(* CoDeSys 2.3.9.41 project: plc_12.pro *)
(* Libraries: STANDARD.LIB 4.10.05 13:14:46, IECSFC.LIB 13.4.06 17:51:28, SYSLIBTIME.LIB 20.2.06 15:31:16, SYSTASKINFO.LIB 20.2.06 15:31:38, ANALYZATION.LIB 5.10.99 11:05:06, SYSLIBCALLBACK.LIB 20.2.06 15:31:08, Util.lib 18.5.10 17:14:28 *)

(* PLC configuration (modules and I/O channels)
Fast discrete inputs [I_SIMPLE_INPUT] node 0, in %IB0 out %QB0 {ChannellName = Fast discrete inputs; Filtrationtime = 1}
  AT %IX0.0 [BitInput] Discrete input 1 {ChannellName = Enter name}
  AT %IX0.1 [BitInput] Discrete input 2 {ChannellName = Enter name}
  AT %IX0.2 [BitInput] Discrete input 3 {ChannellName = Enter name}
  CONTR_PHASE AT %IX0.3 [BitInput] Discrete input 4 {ChannellName = Enter name}
Discrete inputs [ID130] node 1, in %IB1 out %QB1 {ChannellName = Discrete inputs; Filtrationtime_GeneralINP = 0; PinCount = 32}
  AT %IB1.0 [ByteInput] 8 discrete inputs {ChannellName = Enter name}
  AT %IB1.1 [ByteInput] 8 discrete inputs {ChannellName = Enter name}
  AT %IB1.2 [ByteInput] 8 discrete inputs {ChannellName = Enter name}
  AT %IB1.3 [ByteInput] 8 discrete inputs {ChannellName = Enter name}
Fast discrete outputs [OWEN_ID570] node 2, in %IB2 out %QB2 {ChannellName = Fast discrete outputs; SafeValueBool = FALSE; SafeValueBool = FALSE; SafeValueBool = FALSE; SafeValueBool = FALSE; Visibility = No}
  ELV_DROB_RUN AT %QX2.0 [BitOutput] Fast discrete output 1 {ChannellName = Enter name}
  DROB_SHOK_1 AT %QX2.1 [BitOutput] Fast discrete output 2 {ChannellName = Enter name}
  DROB_SHOK_2 AT %QX2.2 [BitOutput] Fast discrete output 3 {ChannellName = Enter name}
  CONV_DROB AT %QX2.3 [BitOutput] Fast discrete output 4 {ChannellName = Enter name}
Discrete outputs [ID131] node 3, in %IB3 out %QB3 {ChannellName = Discrete outputs; SafeValueByte = 0; SafeValueByte = 0; SafeValueByteM = 0; PinCount = 24}
  AT %QB3.0 [ByteOutput] 8 discrete outputs {ChannellName = Enter name}
  AT %QB3.1 [ByteOutput] 8 discrete outputs {ChannellName = Enter name}
  AT %QB3.2 [ByteOutput] 4 discrete outputs {ChannellName = Enter name}
Special input [ID103] node 4, in %IB4 out %QB4 {ChannellName = Special input}
  AT %IX4.0 [BitInput] Special input {ChannellName = Enter name}
Special output [ID104] node 5, in %IB5 out %QB5 {ChannellName = Special output}
  AT %QX5.0 [BitOutput] Special output {ChannellName = Enter name}
AT %QD6.0 [DWordOutput] Last address {ChannellName = Enter name}
AT %QW6.1 [WordOutput] Last error {ChannellName = Enter name}
RS-485-1 [COM1_USART] node 0, in %IB6.0 out %QB6.0 {ChannellName = RS-485-1; CommunicationSpeed = 115200; Parity = NO PARITY CHECK; BitLength = 8 bits; StopLength = One stop bit; InterfaceType = RS485; FrameOriented = RTU; Timeout = 0; Visibility = No}
Universal Modbus device [ID2000] node 1, in %IB6.1 out %QB6.1 {ChannellName = Universal Modbus device; ModuleIP = 10:0:0:223; ServiceTimeout = 150; TCPport = 502; NetMode = Serial; ModuleSlaveAddress = 8; RequestType = By poll time; PeriodOfService = 10; Visibility = No; RepeatCounter = 0; ByteSequence = Trace_mode}
  AT %QB6.1.0 [ComChannel] Command (0xff - Start) {ChannellName = Enter name}
MV8_0 AT %QW6.1.0.0 [WordOutput] {ChannellName = Enter name}
MV8_1 AT %QW6.1.1.0 [WordOutput] {ChannellName = Enter name}
Universal Modbus device [ID2000] node 2, in %IB6.2 out %QB6.2 {ChannellName = Universal Modbus device; ModuleIP = 10:0:0:223; ServiceTimeout = 150; TCPport = 502; NetMode = Serial; ModuleSlaveAddress = 16; RequestType = By poll time; PeriodOfService = 10; Visibility = No; RepeatCounter = 0; ByteSequence = Trace_mode}
  AT %QB6.2.0 [ComChannel] Command (0xff - Start) {ChannellName = Enter name}
MV16_0 AT %QW6.2.0.0 [WordOutput] {ChannellName = Enter name}
MV16_1 AT %QW6.2.1.0 [WordOutput] {ChannellName = Enter name}
Universal Modbus device [ID2000] node 3, in %IB6.3 out %QB6.3 {ChannellName = Universal Modbus device; ModuleIP = 10:0:0:223; ServiceTimeout = 150; TCPport = 502; NetMode = Serial; ModuleSlaveAddress = 24; RequestType = By poll time; PeriodOfService = 10; Visibility = No; RepeatCounter = 0; ByteSequence = Trace_mode}
  AT %QB6.3.0 [ComChannel] Command (0xff - Start) {ChannellName = Enter name}
MV24_0 AT %QW6.3.0.0 [WordOutput] {ChannellName = Enter name}
MV24_1 AT %QW6.3.1.0 [WordOutput] {ChannellName = Enter name}
Universal Modbus device [ID2000] node 4, in %IB6.4 out %QB6.4 {ChannellName = Universal Modbus device; ModuleIP = 10:0:0:223; ServiceTimeout = 150; TCPport = 502; NetMode = Serial; ModuleSlaveAddress = 32; RequestType = By poll time; PeriodOfService = 10; Visibility = No; RepeatCounter = 0; ByteSequence = Trace_mode}
  AT %QB6.4.0 [ComChannel] Command (0xff - Start) {ChannellName = Enter name}
MU01 AT %QW6.4.0.0 [WordOutput] {ChannellName = Enter name}
MU02 AT %QW6.4.1.0 [WordOutput] {ChannellName = Enter name}
MU03 AT %QW6.4.2.0 [WordOutput] {ChannellName = Enter name}
MU04 AT %QW6.4.3.0 [WordOutput] {ChannellName = Enter name}
MU05 AT %QW6.4.4.0 [WordOutput] {ChannellName = Enter name}
MU06 AT %QW6.4.5.0 [WordOutput] {ChannellName = Enter name}
MU07 AT %QW6.4.6.0 [WordOutput] {ChannellName = Enter name}
MU08 AT %QW6.4.7.0 [WordOutput] {ChannellName = Enter name}
MU09 AT %QW6.4.8.0 [WordOutput] {ChannellName = Enter name}
MU10 AT %QW6.4.9.0 [WordOutput] {ChannellName = Enter name}
MU11 AT %QW6.4.10.0 [WordOutput] {ChannellName = Enter name}
MU12 AT %QW6.4.11.0 [WordOutput] {ChannellName = Enter name}
MU13 AT %QW6.4.12.0 [WordOutput] {ChannellName = Enter name}
MU14 AT %QW6.4.13.0 [WordOutput] {ChannellName = Enter name}
MU15 AT %QW6.4.14.0 [WordOutput] {ChannellName = Enter name}
MU16 AT %QW6.4.15.0 [WordOutput] {ChannellName = Enter name}
MU17 AT %QW6.4.16.0 [WordOutput] {ChannellName = Enter name}
MU18 AT %QW6.4.17.0 [WordOutput] {ChannellName = Enter name}
MU19 AT %QW6.4.18.0 [WordOutput] {ChannellName = Enter name}
MU20 AT %QW6.4.19.0 [WordOutput] {ChannellName = Enter name}
MU21 AT %QW6.4.20.0 [WordOutput] {ChannellName = Enter name}
%MMU22 AT %QW6.4.21.0 [WordOutput] {ChannellName = Enter name}
MU23 AT %QW6.4.22.0 [WordOutput] {ChannellName = Enter name}
MU24 AT %QW6.4.23.0 [WordOutput] {ChannellName = Enter name}
MU25 AT %QW6.4.24.0 [WordOutput] {ChannellName = Enter name}
MU26 AT %QW6.4.25.0 [WordOutput] {ChannellName = Enter name}
MU27 AT %QW6.4.26.0 [WordOutput] {ChannellName = Enter name}
MU28 AT %QW6.4.27.0 [WordOutput] {ChannellName = Enter name}
MU29 AT %QW6.4.28.0 [WordOutput] {ChannellName = Enter name}
MU30 AT %QW6.4.29.0 [WordOutput] {ChannellName = Enter name}
MU31 AT %QW6.4.30.0 [WordOutput] {ChannellName = Enter name}
MU32 AT %QW6.4.31.0 [WordOutput] {ChannellName = Enter name}
AT %QB6.5.0 [ComChannel] Command (0xff - Start) {ChannellName = Enter name}
ELV_CURRENT_4 AT %QW6.5.0.0 [WordOutput] {ChannellName = Enter name}
SHNK_CURRENT_4 AT %QW6.5.1.0 [WordOutput] {ChannellName = Enter name}
MILL_SUCTION_4 AT %QW6.5.2.0 [WordOutput] {ChannellName = Enter name}
SHNK_CURRENT_3 AT %QW6.5.3.0 [WordOutput] {ChannellName = Enter name}
MILL_SUCTION_3 AT %QW6.5.4.0 [WordOutput] {ChannellName = Enter name}
TCP [TCP_ID221] node 0, in %IB7.0.0 out %QB7.0.0 {ChannellName = TCP; RemotePort = 502; Visibility = No}
TCP [TCP_ID221] node 1, in %IB7.0.1 out %QB7.0.1 {ChannellName = TCP; RemotePort = 503; Visibility = No}
CONV_1_DIO AT %QW7.1.0 [WordOutput] {ChannellName = Enter name}
CONV_1_CURRENT AT %QW7.2.0 [WordOutput] {ChannellName = Enter name}
CONV_1_FREQ AT %QW7.3.0 [WordOutput] {ChannellName = Enter name}
CONV_1_SETPOINT AT %QW7.4.0 [WordOutput] {ChannellName = Enter name}
CONV_1_wHOUR AT %QW7.5.0 [WordOutput] {ChannellName = Enter name}
CONV_1_stopTIME AT %QW7.6.0 [WordOutput] {ChannellName = Enter name}
CONV_1_startTIME AT %QW7.7.0 [WordOutput] {ChannellName = Enter name}
CONV_1_stopTIME_W AT %QW7.8.0 [WordOutput] {ChannellName = Enter name}
CONV_1_startTIME_W AT %QW7.9.0 [WordOutput] {ChannellName = Enter name}
FAN_1_DIO AT %QW7.10.0 [WordOutput] {ChannellName = Enter name}
FAN_1_CURRENT AT %QW7.11.0 [WordOutput] {ChannellName = Enter name}
FAN_1_FREQ AT %QW7.12.0 [WordOutput] {ChannellName = Enter name}
FAN_1_SETPOINT AT %QW7.13.0 [WordOutput] {ChannellName = Enter name}
FAN_1_SUCTION AT %QW7.14.0 [WordOutput] {ChannellName = Enter name}
FAN_1_wHOUR AT %QW7.15.0 [WordOutput] {ChannellName = Enter name}
FAN_1_stopTIME AT %QW7.16.0 [WordOutput] {ChannellName = Enter name}
FAN_1_startTIME AT %QW7.17.0 [WordOutput] {ChannellName = Enter name}
FAN_1_stopTIME_W AT %QW7.18.0 [WordOutput] {ChannellName = Enter name}
FAN_1_startTIME_W AT %QW7.19.0 [WordOutput] {ChannellName = Enter name}
MILL_1_DIO AT %QW7.20.0 [WordOutput] {ChannellName = Enter name}
MILL_1_CURRENT AT %QW7.21.0 [WordOutput] {ChannellName = Enter name}
MILL_1_FREQ AT %QW7.22.0 [WordOutput] {ChannellName = Enter name}
MILL_1_SETPOINT AT %QW7.23.0 [WordOutput] {ChannellName = Enter name}
MILL_1_wHOUR AT %QW7.24.0 [WordOutput] {ChannellName = Enter name}
MILL_1_stopTIME AT %QW7.25.0 [WordOutput] {ChannellName = Enter name}
MILL_1_startTIME AT %QW7.26.0 [WordOutput] {ChannellName = Enter name}
MILL_1_stopTIME_W AT %QW7.27.0 [WordOutput] {ChannellName = Enter name}
MILL_1_startTIME_W AT %QW7.28.0 [WordOutput] {ChannellName = Enter name}
SEP_1_DIO AT %QW7.29.0 [WordOutput] {ChannellName = Enter name}
SEP_1_CURRENT AT %QW7.30.0 [WordOutput] {ChannellName = Enter name}
SEP_1_FREQ AT %QW7.31.0 [WordOutput] {ChannellName = Enter name}
SEP_1_SETPOINT AT %QW7.32.0 [WordOutput] {ChannellName = Enter name}
SEP_1_wHOUR AT %QW7.33.0 [WordOutput] {ChannellName = Enter name}
SEP_1_stopTIME AT %QW7.34.0 [WordOutput] {ChannellName = Enter name}
SEP_1_startTIME AT %QW7.35.0 [WordOutput] {ChannellName = Enter name}
SEP_1_stopTIME_W AT %QW7.36.0 [WordOutput] {ChannellName = Enter name}
SEP_1_startTIME_W AT %QW7.37.0 [WordOutput] {ChannellName = Enter name}
2 byte [Register] node 38, in %IB7.38 out %QB7.38 {ChannellName = 2 byte}
  CONV_2_DIO AT %QW7.38.0 [WordOutput] {ChannellName = Enter name}
2 byte [Register] node 39, in %IB7.39 out %QB7.39 {ChannellName = 2 byte}
  CONV_2_CURRENT AT %QW7.39.0 [WordOutput] {ChannellName = Enter name}
2 byte [Register] node 40, in %IB7.40 out %QB7.40 {ChannellName = 2 byte}
  CONV_2_FREQ AT %QW7.40.0 [WordOutput] {ChannellName = Enter name}
2 byte [Register] node 41, in %IB7.41 out %QB7.41 {ChannellName = 2 byte}
  CONV_2_SETPOINT AT %QW7.41.0 [WordOutput] {ChannellName = Enter name}
  CONV_2_wHOUR AT %QW7.42.0 [WordOutput] {ChannellName = Enter name}
  CONV_2_stopTIME AT %QW7.43.0 [WordOutput] {ChannellName = Enter name}
  CONV_2_startTIME AT %QW7.44.0 [WordOutput] {ChannellName = Enter name}
  CONV_2_stopTIME_W AT %QW7.45.0 [WordOutput] {ChannellName = Enter name}
2 byte [Register] node 46, in %IB7.46 out %QB7.46 {ChannellName = 2 byte}
  CONV_2_startTIME_W AT %QW7.46.0 [WordOutput] {ChannellName = Enter name}
2 byte [Register] node 47, in %IB7.47 out %QB7.47 {ChannellName = 2 byte}
  FAN_2_DIO AT %QW7.47.0 [WordOutput] {ChannellName = Enter name}
2 byte [Register] node 48, in %IB7.48 out %QB7.48 {ChannellName = 2 byte}
  FAN_2_CURRENT AT %QW7.48.0 [WordOutput] {ChannellName = Enter name}
2 byte [Register] node 49, in %IB7.49 out %QB7.49 {ChannellName = 2 byte}
  FAN_2_FREQ AT %QW7.49.0 [WordOutput] {ChannellName = Enter name}
  FAN_2_SETPOINT AT %QW7.50.0 [WordOutput] {ChannellName = Enter name}
  FAN_2_SUCTION AT %QW7.51.0 [WordOutput] {ChannellName = Enter name}
  FAN_2_wHOUR AT %QW7.52.0 [WordOutput] {ChannellName = Enter name}
  FAN_2_stopTIME AT %QW7.53.0 [WordOutput] {ChannellName = Enter name}
  FAN_2_startTIME AT %QW7.54.0 [WordOutput] {ChannellName = Enter name}
2 byte [Register] node 55, in %IB7.55 out %QB7.55 {ChannellName = 2 byte}
  FAN_2_stopTIME_W AT %QW7.55.0 [WordOutput] {ChannellName = Enter name}
  FAN_2_startTIME_W AT %QW7.56.0 [WordOutput] {ChannellName = Enter name}
2 byte [Register] node 57, in %IB7.57 out %QB7.57 {ChannellName = 2 byte}
  MILL_2_DIO AT %QW7.57.0 [WordOutput] {ChannellName = Enter name}
  MILL_2_CURRENT AT %QW7.58.0 [WordOutput] {ChannellName = Enter name}
  MILL_2_FREQ AT %QW7.59.0 [WordOutput] {ChannellName = Enter name}
  MILL_2_SETPOINT AT %QW7.60.0 [WordOutput] {ChannellName = Enter name}
2 byte [Register] node 61, in %IB7.61 out %QB7.61 {ChannellName = 2 byte}
  MILL_2_wHOUR AT %QW7.61.0 [WordOutput] {ChannellName = Enter name}
  MILL_2_stopTIME AT %QW7.62.0 [WordOutput] {ChannellName = Enter name}
2 byte [Register] node 63, in %IB7.63 out %QB7.63 {ChannellName = 2 byte}
  MILL_2_startTIME AT %QW7.63.0 [WordOutput] {ChannellName = Enter name}
  MILL_2_stopTIME_W AT %QW7.64.0 [WordOutput] {ChannellName = Enter name}
2 byte [Register] node 65, in %IB7.65 out %QB7.65 {ChannellName = 2 byte}
  MILL_2_startTIME_W AT %QW7.65.0 [WordOutput] {ChannellName = Enter name}
2 byte [Register] node 66, in %IB7.66 out %QB7.66 {ChannellName = 2 byte}
  SEP_2_DIO AT %QW7.66.0 [WordOutput] {ChannellName = Enter name}
  SEP_2_CURRENT AT %QW7.67.0 [WordOutput] {ChannellName = Enter name}
2 byte [Register] node 68, in %IB7.68 out %QB7.68 {ChannellName = 2 byte}
  SEP_2_FREQ AT %QW7.68.0 [WordOutput] {ChannellName = Enter name}
  SEP_2_SETPOINT AT %QW7.69.0 [WordOutput] {ChannellName = Enter name}
2 byte [Register] node 70, in %IB7.70 out %QB7.70 {ChannellName = 2 byte}
  SEP_2_wHOUR AT %QW7.70.0 [WordOutput] {ChannellName = Enter name}
2 byte [Register] node 71, in %IB7.71 out %QB7.71 {ChannellName = 2 byte}
  SEP_2_stopTIME AT %QW7.71.0 [WordOutput] {ChannellName = Enter name}
2 byte [Register] node 72, in %IB7.72 out %QB7.72 {ChannellName = 2 byte}
  SEP_2_startTIME AT %QW7.72.0 [WordOutput] {ChannellName = Enter name}
  SEP_2_stopTIME_W AT %QW7.73.0 [WordOutput] {ChannellName = Enter name}
2 byte [Register] node 74, in %IB7.74 out %QB7.74 {ChannellName = 2 byte}
  SEP_2_startTIME_W AT %QW7.74.0 [WordOutput] {ChannellName = Enter name}
  ELEV_12_DIO AT %QW7.75.0 [WordOutput] {ChannellName = Enter name}
2 byte [Register] node 76, in %IB7.76 out %QB7.76 {ChannellName = 2 byte}
  ELEV_12_CURRENT AT %QW7.76.0 [WordOutput] {ChannellName = Enter name}
2 byte [Register] node 77, in %IB7.77 out %QB7.77 {ChannellName = 2 byte}
  ELEV_12_wHOUR AT %QW7.77.0 [WordOutput] {ChannellName = Enter name}
  ELEV_12_stopTIME AT %QW7.78.0 [WordOutput] {ChannellName = Enter name}
2 byte [Register] node 79, in %IB7.79 out %QB7.79 {ChannellName = 2 byte}
  ELEV_12_startTIME AT %QW7.79.0 [WordOutput] {ChannellName = Enter name}
  ELEV_12_stopTIME_W AT %QW7.80.0 [WordOutput] {ChannellName = Enter name}
  ELEV_12_startTIME_W AT %QW7.81.0 [WordOutput] {ChannellName = Enter name}
  SHNEK_1_DIO AT %QW7.82.0 [WordOutput] {ChannellName = Enter name}
  SHNEK_1_CURRENT AT %QW7.83.0 [WordOutput] {ChannellName = Enter name}
  SHNEK_1_wHOUR AT %QW7.84.0 [WordOutput] {ChannellName = Enter name}
  SHNEK_1_stopTIME AT %QW7.85.0 [WordOutput] {ChannellName = Enter name}
  SHNEK_1_startTIME AT %QW7.86.0 [WordOutput] {ChannellName = Enter name}
2 byte [Register] node 87, in %IB7.87 out %QB7.87 {ChannellName = 2 byte}
  SHNEK_1_stopTIME_W AT %QW7.87.0 [WordOutput] {ChannellName = Enter name}
2 byte [Register] node 88, in %IB7.88 out %QB7.88 {ChannellName = 2 byte}
  SHNEK_1_startTIME_W AT %QW7.88.0 [WordOutput] {ChannellName = Enter name}
2 byte [Register] node 89, in %IB7.89 out %QB7.89 {ChannellName = 2 byte}
  SHNEK_2_DIO AT %QW7.89.0 [WordOutput] {ChannellName = Enter name}
2 byte [Register] node 90, in %IB7.90 out %QB7.90 {ChannellName = 2 byte}
  SHNEK_2_CURRENT AT %QW7.90.0 [WordOutput] {ChannellName = Enter name}
2 byte [Register] node 91, in %IB7.91 out %QB7.91 {ChannellName = 2 byte}
  SHNEK_2_wHOUR AT %QW7.91.0 [WordOutput] {ChannellName = Enter name}
2 byte [Register] node 92, in %IB7.92 out %QB7.92 {ChannellName = 2 byte}
  SHNEK_2_stopTIME AT %QW7.92.0 [WordOutput] {ChannellName = Enter name}
2 byte [Register] node 93, in %IB7.93 out %QB7.93 {ChannellName = 2 byte}
  SHNEK_2_startTIME AT %QW7.93.0 [WordOutput] {ChannellName = Enter name}
  SHNEK_2_stopTIME_W AT %QW7.94.0 [WordOutput] {ChannellName = Enter name}
2 byte [Register] node 95, in %IB7.95 out %QB7.95 {ChannellName = 2 byte}
  SHNEK_2_startTIME_W AT %QW7.95.0 [WordOutput] {ChannellName = Enter name}
2 byte [Register] node 96, in %IB7.96 out %QB7.96 {ChannellName = 2 byte}
  STAR_11_DIO AT %QW7.96.0 [WordOutput] {ChannellName = Enter name}
  STAR_11_wHOUR AT %QW7.97.0 [WordOutput] {ChannellName = Enter name}
  STAR_11_stopTIME AT %QW7.98.0 [WordOutput] {ChannellName = Enter name}
  STAR_11_startTIME AT %QW7.99.0 [WordOutput] {ChannellName = Enter name}
  STAR_11_stopTIME_W AT %QW7.100.0 [WordOutput] {ChannellName = Enter name}
  STAR_11_startTIME_W AT %QW7.101.0 [WordOutput] {ChannellName = Enter name}
  STAR_12_DIO AT %QW7.102.0 [WordOutput] {ChannellName = Enter name}
  STAR_12_wHOUR AT %QW7.103.0 [WordOutput] {ChannellName = Enter name}
  STAR_12_stopTIME AT %QW7.104.0 [WordOutput] {ChannellName = Enter name}
  STAR_12_startTIME AT %QW7.105.0 [WordOutput] {ChannellName = Enter name}
  STAR_12_stopTIME_W AT %QW7.106.0 [WordOutput] {ChannellName = Enter name}
  STAR_12_startTIME_W AT %QW7.107.0 [WordOutput] {ChannellName = Enter name}
  STAR_21_DIO AT %QW7.108.0 [WordOutput] {ChannellName = Enter name}
  STAR_21_wHOUR AT %QW7.109.0 [WordOutput] {ChannellName = Enter name}
  STAR_21_stopTIME AT %QW7.110.0 [WordOutput] {ChannellName = Enter name}
  STAR_21_startTIME AT %QW7.111.0 [WordOutput] {ChannellName = Enter name}
  STAR_21_stopTIME_W AT %QW7.112.0 [WordOutput] {ChannellName = Enter name}
  STAR_21_startTIME_W AT %QW7.113.0 [WordOutput] {ChannellName = Enter name}
  STAR_22_DIO AT %QW7.114.0 [WordOutput] {ChannellName = Enter name}
  STAR_22_wHOUR AT %QW7.115.0 [WordOutput] {ChannellName = Enter name}
  STAR_22_stopTIME AT %QW7.116.0 [WordOutput] {ChannellName = Enter name}
  STAR_22_startTIME AT %QW7.117.0 [WordOutput] {ChannellName = Enter name}
  STAR_22_stopTIME_W AT %QW7.118.0 [WordOutput] {ChannellName = Enter name}
  STAR_22_startTIME_W AT %QW7.119.0 [WordOutput] {ChannellName = Enter name}
  OIL_1_DIO AT %QW7.120.0 [WordOutput] {ChannellName = Enter name}
  OIL_1_wHOUR AT %QW7.121.0 [WordOutput] {ChannellName = Enter name}
  OIL_1_stopTIME AT %QW7.122.0 [WordOutput] {ChannellName = Enter name}
  OIL_1_startTIME AT %QW7.123.0 [WordOutput] {ChannellName = Enter name}
  OIL_1_stopTIME_W AT %QW7.124.0 [WordOutput] {ChannellName = Enter name}
  OIL_1_startTIME_W AT %QW7.125.0 [WordOutput] {ChannellName = Enter name}
  OIL_2_DIO AT %QW7.126.0 [WordOutput] {ChannellName = Enter name}
  OIL_2_wHOUR AT %QW7.127.0 [WordOutput] {ChannellName = Enter name}
  OIL_2_stopTIME AT %QW7.128.0 [WordOutput] {ChannellName = Enter name}
  OIL_2_startTIME AT %QW7.129.0 [WordOutput] {ChannellName = Enter name}
  OIL_2_stopTIME_W AT %QW7.130.0 [WordOutput] {ChannellName = Enter name}
  OIL_2_startTIME_W AT %QW7.131.0 [WordOutput] {ChannellName = Enter name}
  VIBR_1_DIO AT %QW7.132.0 [WordOutput] {ChannellName = Enter name}
  VIBR_2_DIO AT %QW7.133.0 [WordOutput] {ChannellName = Enter name}
  SHNK_SIKL_1_DIO AT %QW7.134.0 [WordOutput] {ChannellName = Enter name}
  SHNK_SIKL_1_wHOUR AT %QW7.135.0 [WordOutput] {ChannellName = Enter name}
  SHNK_SIKL_1_stopTIME AT %QW7.136.0 [WordOutput] {ChannellName = Enter name}
  SHNK_SIKL_1_startTIME AT %QW7.137.0 [WordOutput] {ChannellName = Enter name}
  SHNK_SIKL_1_stopTIME_W AT %QW7.138.0 [WordOutput] {ChannellName = Enter name}
  SHNK_SIKL_1_startTIME_W AT %QW7.139.0 [WordOutput] {ChannellName = Enter name}
  SHNK_SIKL_2_DIO AT %QW7.140.0 [WordOutput] {ChannellName = Enter name}
  SHNK_SIKL_2_wHOUR AT %QW7.141.0 [WordOutput] {ChannellName = Enter name}
  SHNK_SIKL_2_stopTIME AT %QW7.142.0 [WordOutput] {ChannellName = Enter name}
  SHNK_SIKL_2_startTIME AT %QW7.143.0 [WordOutput] {ChannellName = Enter name}
  SHNK_SIKL_2_stopTIME_W AT %QW7.144.0 [WordOutput] {ChannellName = Enter name}
  SHNK_SIKL_2_startTIME_W AT %QW7.145.0 [WordOutput] {ChannellName = Enter name}
  VALV_1_DIO AT %QW7.146.0 [WordOutput] {ChannellName = Enter name}
  VALV_2_DIO AT %QW7.147.0 [WordOutput] {ChannellName = Enter name}
  TANK_12_DIO AT %QW7.148.0 [WordOutput] {ChannellName = Enter name}
  HORN_12_DIO AT %QW7.149.0 [WordOutput] {ChannellName = Enter name}
  MILL_1 AT %QW7.150.0 [WordOutput] {ChannellName = Enter name}
  MILL_2 AT %QW7.151.0 [WordOutput] {ChannellName = Enter name}
ModBus (Master) [MODBUS_MASTER_ID450] node 8, in %IB8 out %QB8 {ChannellName = ModBus (Master); Visibility = No}
  AT %QD8.0 [DWordOutput] Last address {ChannellName = Enter name}
  AT %QW8.1 [WordOutput] Last error {ChannellName = Enter name}
  RS-485-2 [COM3_USART] node 0, in %IB8.0 out %QB8.0 {ChannellName = RS-485-2; CommunicationSpeed = 57600; Parity = NO PARITY CHECK; BitLength = 8 bits; StopLength = One stop bit; InterfaceType = RS485; FrameOriented = RTU; Timeout = 50; Visibility = No}
  Universal Modbus device [ID2000] node 1, in %IB8.1 out %QB8.1 {ChannellName = Universal Modbus device; ModuleIP = 10:0:0:223; ServiceTimeout = 150; TCPport = 502; NetMode = Serial; ModuleSlaveAddress = 1; RequestType = By poll time; PeriodOfService = 100; Visibility = No; RepeatCounter = 0; ByteSequence = Trace_mode}
    AT %QB8.1.0 [ComChannel] Command (0xff - Start) {ChannellName = Enter name}
CONV_PANEL_1 AT %QW8.1.0.0 [WordOutput] {ChannellName = Enter name}
CONV_FREQ_1 AT %QW8.1.1.0 [WordOutput] {ChannellName = Enter name}
CONV_CURRENT_1 AT %QW8.1.2.0 [WordOutput] {ChannellName = Enter name}
CONV_SET_FREQ_1 AT %QW8.1.3.0 [WordOutput] {ChannellName = Enter name}
AT %QB8.2.0 [ComChannel] Command (0xff - Start) {ChannellName = Enter name}
FAN_PANEL_1 AT %QW8.2.0.0 [WordOutput] {ChannellName = Enter name}
FAN_FREQ_1 AT %QW8.2.1.0 [WordOutput] {ChannellName = Enter name}
FAN_CURRENT_1 AT %QW8.2.2.0 [WordOutput] {ChannellName = Enter name}
FAN_SET_FREQ_1 AT %QW8.2.3.0 [WordOutput] {ChannellName = Enter name}
AT %QB8.3.0 [ComChannel] Command (0xff - Start) {ChannellName = Enter name}
MILL_PANEL_1 AT %QW8.3.0.0 [WordOutput] {ChannellName = Enter name}
MILL_FREQ_1 AT %QW8.3.1.0 [WordOutput] {ChannellName = Enter name}
MILL_CURRENT_1 AT %QW8.3.2.0 [WordOutput] {ChannellName = Enter name}
MILL_SET_FREQ_1 AT %QW8.3.3.0 [WordOutput] {ChannellName = Enter name}
AT %QB8.4.0 [ComChannel] Command (0xff - Start) {ChannellName = Enter name}
SEP_PANEL_1 AT %QW8.4.0.0 [WordOutput] {ChannellName = Enter name}
SEP_FREQ_1 AT %QW8.4.1.0 [WordOutput] {ChannellName = Enter name}
SEP_CURRENT_1 AT %QW8.4.2.0 [WordOutput] {ChannellName = Enter name}
SEP_SET_FREQ_1 AT %QW8.4.3.0 [WordOutput] {ChannellName = Enter name}
AT %QB8.5.0 [ComChannel] Command (0xff - Start) {ChannellName = Enter name}
CONV_PANEL_2 AT %QW8.5.0.0 [WordOutput] {ChannellName = Enter name}
CONV_FREQ_2 AT %QW8.5.1.0 [WordOutput] {ChannellName = Enter name}
CONV_CURRENT_2 AT %QW8.5.2.0 [WordOutput] {ChannellName = Enter name}
CONV_SET_FREQ_2 AT %QW8.5.3.0 [WordOutput] {ChannellName = Enter name}
AT %QB8.6.0 [ComChannel] Command (0xff - Start) {ChannellName = Enter name}
FAN_PANEL_2 AT %QW8.6.0.0 [WordOutput] {ChannellName = Enter name}
FAN_FREQ_2 AT %QW8.6.1.0 [WordOutput] {ChannellName = Enter name}
FAN_CURRENT_2 AT %QW8.6.2.0 [WordOutput] {ChannellName = Enter name}
FAN_SET_FREQ_2 AT %QW8.6.3.0 [WordOutput] {ChannellName = Enter name}
Universal Modbus device [ID2000] node 7, in %IB8.7 out %QB8.7 {ChannellName = Universal Modbus device; ModuleIP = 10:0:0:223; ServiceTimeout = 150; TCPport = 502; NetMode = Serial; ModuleSlaveAddress = 7; RequestType = By poll time; PeriodOfService = 100; Visibility = No; RepeatCounter = 0; ByteSequence = Trace_mode}
  AT %QB8.7.0 [ComChannel] Command (0xff - Start) {ChannellName = Enter name}
MILL_PANEL_2 AT %QW8.7.0.0 [WordOutput] {ChannellName = Enter name}
MILL_FREQ_2 AT %QW8.7.1.0 [WordOutput] {ChannellName = Enter name}
MILL_CURRENT_2 AT %QW8.7.2.0 [WordOutput] {ChannellName = Enter name}
MILL_SET_FREQ_2 AT %QW8.7.3.0 [WordOutput] {ChannellName = Enter name}
Universal Modbus device [ID2000] node 8, in %IB8.8 out %QB8.8 {ChannellName = Universal Modbus device; ModuleIP = 10:0:0:223; ServiceTimeout = 150; TCPport = 502; NetMode = Serial; ModuleSlaveAddress = 8; RequestType = By poll time; PeriodOfService = 100; Visibility = No; RepeatCounter = 0; ByteSequence = Trace_mode}
  AT %QB8.8.0 [ComChannel] Command (0xff - Start) {ChannellName = Enter name}
SEP_PANEL_2 AT %QW8.8.0.0 [WordOutput] {ChannellName = Enter name}
SEP_FREQ_2 AT %QW8.8.1.0 [WordOutput] {ChannellName = Enter name}
SEP_CURRENT_2 AT %QW8.8.2.0 [WordOutput] {ChannellName = Enter name}
SEP_SET_FREQ_2 AT %QW8.8.3.0 [WordOutput] {ChannellName = Enter name}
*)

(* Global variable list: Global_Variables *)
VAR_GLOBAL
	kvitVaqt : TIME := T#60s;
	tpKVIT : TP;
	TANK_MAX : BOOL;
	(*MU 32 DISCRET OUTPUT*)
	ELV_RUN : BOOL;			(*DO01*)
	SHNK_RUN_2  : BOOL;		(*DO02*)
	SHNK_SKL_RUN_2  : BOOL;	(*DO03*)
	STAR_RUN_21  : BOOL;		(*DO04*)
	STAR_RUN_22  : BOOL;		(*DO05*)
	SEPR_RUN_2  : BOOL;		(*DO06*)
	OIL_ST_RUN_2  : BOOL;		(*DO07*)
	MILL_RUN_2  : BOOL;		(*DO08*)
	FAN_RUN_2  : BOOL;		(*DO09*)
	CONV_RUN_2  : BOOL;		(*DO10*)
	VIBR_RUN_2  : BOOL;		(*DO11*)
	VALV_RUN_2 : BOOL;		(*DO12*)
	HORN_RUN_2 : BOOL; 		(*DO13*)

	(*ELV_RUN_3 :  BOOL ; 		DO17*)
	SHNK_RUN_1 :  BOOL ; 		(*DO18*)
	SHNK_SKL_RUN_1 :  BOOL ; (*DO19*)
	STAR_RUN_11 :  BOOL ;  	(*DO20*)
	STAR_RUN_12 :  BOOL ;  	(*DO21*)
	SEPR_RUN_1 :  BOOL ;  		(*DO22*)
	OIL_ST_RUN_1 :  BOOL ;  	(*DO23*)
	MILL_RUN_1 :  BOOL ;  		(*DO24*)
	FAN_RUN_1 :  BOOL ;  		(*DO25*)
	CONV_RUN_1 :  BOOL ; 		(*DO26*)
	VIBR_RUN_1 :  BOOL ;  		(*DO27*)
	VALV_RUN_1 :  BOOL ;  		(*DO28*)
	HORN_RUN_1 :  BOOL ; 		(*DO29*)
	(*MU 32 DISCRET OUTPUT*)
	(*MV 24 DISCRET INPUT*)
	ELV_KM  : BOOL;				(*DI01*)
	SHNK_KM_2  : BOOL;			(*DI02*)
	SHNK_SKL_KM_2  : BOOL;		(*DI03*)
	STAR_KM_21  : BOOL;			(*DI04*)
	STAR_KM_22  : BOOL;			(*DI05*)
	SEPR_KM_2  : BOOL;			(*DI06*)
	OIL_ST_KM_2  : BOOL;			(*DI07*)
	MILL_KM_2  : BOOL;			(*DI08*)
	MATER_FULL_2  : BOOL;		(*DI09*)
	FAN_KM_2  : BOOL;				(*DI10*)
	CONV_KM_2  : BOOL;			(*DI11*)
	VIBR_KM_2  : BOOL;			(*DI12*)

				(*DI17*)
	SHNK_KM_1  : BOOL;			(*DI18*)
	SHNK_SKL_KM_1  : BOOL;		(*DI19*)
	STAR_KM_11  : BOOL;			(*DI20*)
	STAR_KM_12  : BOOL;			(*DI21*)
	SEPR_KM_1  : BOOL;			(*DI22*)
	OIL_ST_KM_1  : BOOL;			(*DI23*)
	MILL_KM_1  : BOOL;			(*DI24*)
	MATER_FULL_1  : BOOL;		(*DI25*)
	FAN_KM_1  : BOOL;				(*DI26*)
	CONV_KM_1  : BOOL;			(*DI27*)
	VIBR_KM_1  : BOOL;			(*DI28*)
	(*MV 24 DISCRET INPUT*)
	(*MV 16 DISCRET INPUT*)
	ELV_STOP_1  : BOOL;			(*DI01*)
	SHNK_STOP_1  : BOOL;			(*DI02*)
	SHNK_SKL_STOP_1  : BOOL;	(*DI03*)
	STAR_STOP_11  : BOOL;		(*DI04*)
	STAR_STOP_12  : BOOL;		(*DI05*)
	SEPR_STOP_1  : BOOL;			(*DI06*)
	OIL_ST_STOP_1  : BOOL;		(*DI07*)
	MILL_STOP_1  : BOOL;			(*DI08*)
	FAN_STOP_1  : BOOL;			(*DI09*)
	CONV_STOP_1  : BOOL;			(*DI10*)
	VIBR_STOP_1  : BOOL;			(*DI11*)

	ELV_START_1 : BOOL;			(*DI17*)
	SHNK_START_1 : BOOL;			(*DI18*)
	SHNK_SKL_START_1 : BOOL;	(*DI19*)
	STAR_START_11 : BOOL;		(*DI20*)
	STAR_START_12 : BOOL;		(*DI21*)
	SEPR_START_1 : BOOL;			(*DI22*)
	OIL_ST_START_1 : BOOL;		(*DI23*)
	MILL_START_1 : BOOL;			(*DI24*)
	FAN_START_1 : BOOL;			(*DI25*)
	CONV_START_1 : BOOL;		(*DI26*)
	VIBR_START_1 : BOOL;			(*DI27*)
	(*MV 16 DISCRET INPUT*)
	(*MV 08 DISCRET INPUT*)
	ELV_STOP_2  : BOOL;			(*DI01*)
	SHNK_STOP_2  : BOOL;			(*DI02*)
	SHNK_SKL_STOP_2  : BOOL;	(*DI03*)
	STAR_STOP_21  : BOOL;		(*DI04*)
	STAR_STOP_22  : BOOL;		(*DI05*)
	SEPR_STOP_2  : BOOL;			(*DI06*)
	OIL_ST_STOP_2  : BOOL;		(*DI07*)
	MILL_STOP_2  : BOOL;			(*DI08*)
	FAN_STOP_2  : BOOL;			(*DI09*)
	CONV_STOP_2  : BOOL;			(*DI10*)
	VIBR_STOP_2  : BOOL;			(*DI11*)

	ELV_START_2  : BOOL;			(*DI17*)
	SHNK_START_2  : BOOL;		(*DI18*)
	SHNK_SKL_START_2  : BOOL;	(*DI19*)
	STAR_START_21  : BOOL;		(*DI20*)
	STAR_START_22  : BOOL;		(*DI21*)
	SEPR_START_2  : BOOL;		(*DI22*)
	OIL_ST_START_2  : BOOL;		(*DI23*)
	MILL_START_2  : BOOL;			(*DI24*)
	FAN_START_2  : BOOL;			(*DI25*)
	CONV_START_2  : BOOL;			(*DI26*)
	VIBR_START_2  : BOOL;			(*DI27*)
	(*MV 08 DISCRET INPUT*)
END_VAR

(* POU PLC_PRG, ST *)
PROGRAM PLC_PRG
VAR
END_VAR
main();
ALARMS();
RESET_ALRM();
TRANSLATE();
END_PROGRAM

(* POU main, LD *)
PROGRAM main
VAR
	MAH_YET1: BOOL;
	VAQT : TIME := T#6s;
	vaqtInduc : WORD := 15;
	VIBRATOR1_T: BOOL;
	TON1: TON;
	TON2: TON;
	OUT: BOOL;

	STOP: BOOL;
	CHIQSH: BOOL;
	PUSK: BOOL;
	MAH_YET2: BOOL;
	VIBRATOR2_T: BOOL;
	induk: BOOL;

	ALR_ELEV1: BOOL;
	ALR_ELEV2: BOOL;
	ALR_ELEV3: BOOL;
	ALR_ELEV4: BOOL;
	EL_12: ELEV;
	SHNK1: SHNEK;
	SHNK2: SHNEK;
	SHNEK_SIKL1: SHNEK_SIKL;
	SHNEK_SIKL2: SHNEK_SIKL;
	STAR_11: STAR_1;
	STAR_21: STAR_1;
	STAR_12: STAR_2;
	STAR_22: STAR_2;
	SEP1: SEP;
	SEP2: SEP;
	OIL1: OIL;
	MILL1: MILL
;
	OIL2: OIL;
	MILL2: MILL;
	FAN1: FAN;
	FAN2: FAN;
	CONV1: CONV;
	CONV2: CONV;

	test: BOOL;
	test1: BOOL;
	test3: BOOL;
	TEST2: BOOL;
	TEST4: BOOL;
	ELV_RUN2: BOOL;
END_VAR
VAR (* helpers for the ST form of the networks *)
	_p1 : BOOL;
	_p2 : BOOL;
END_VAR
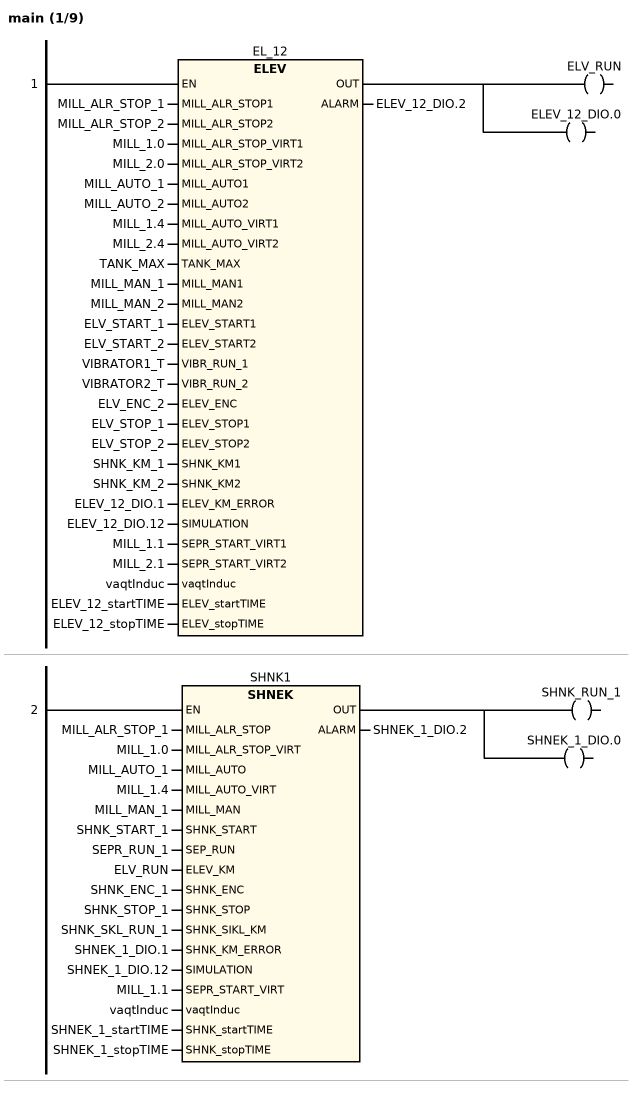
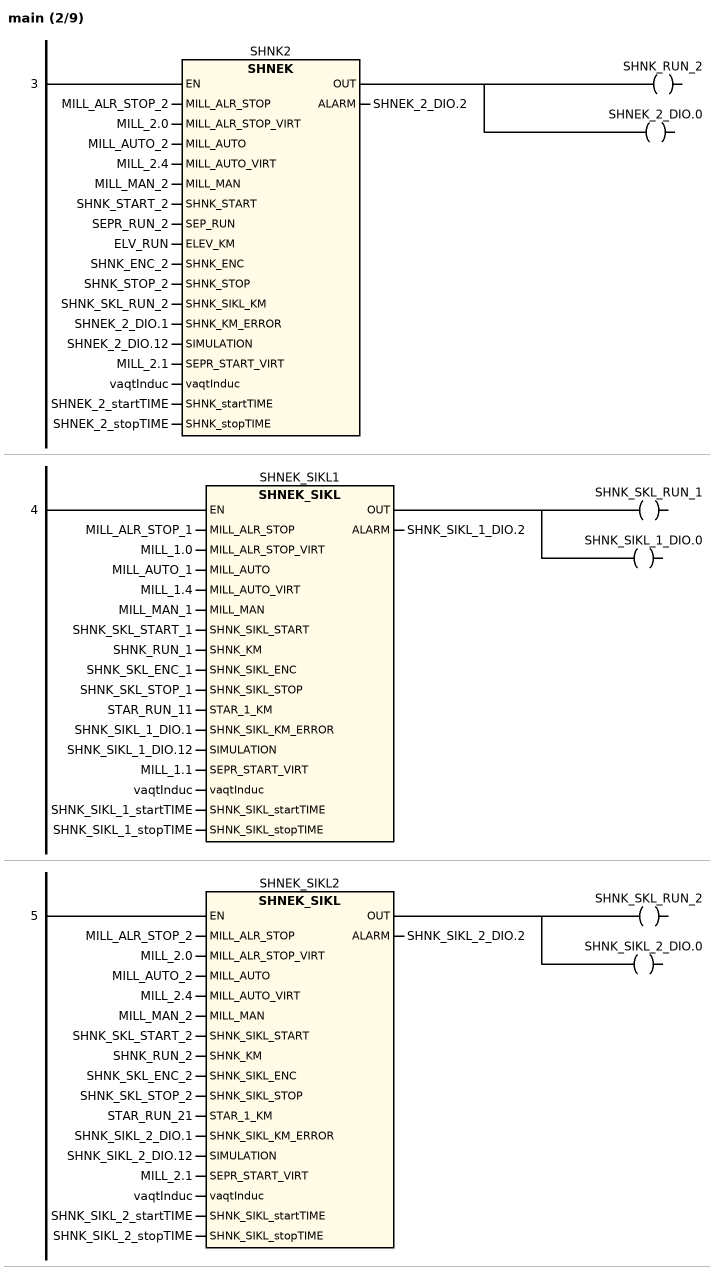
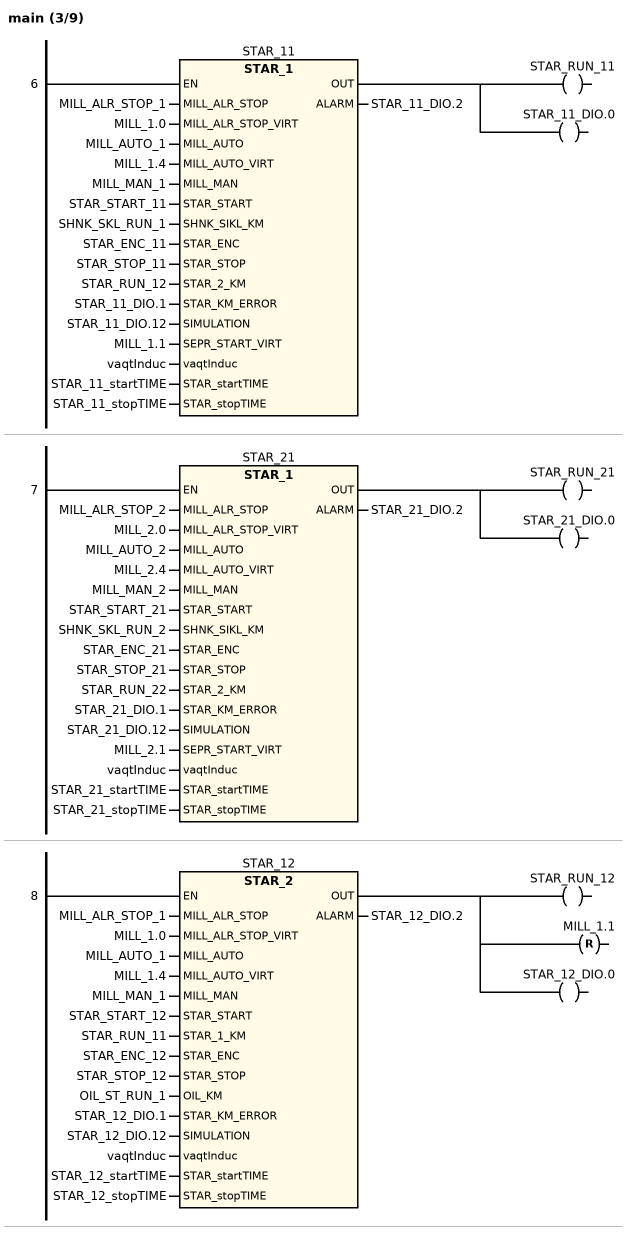
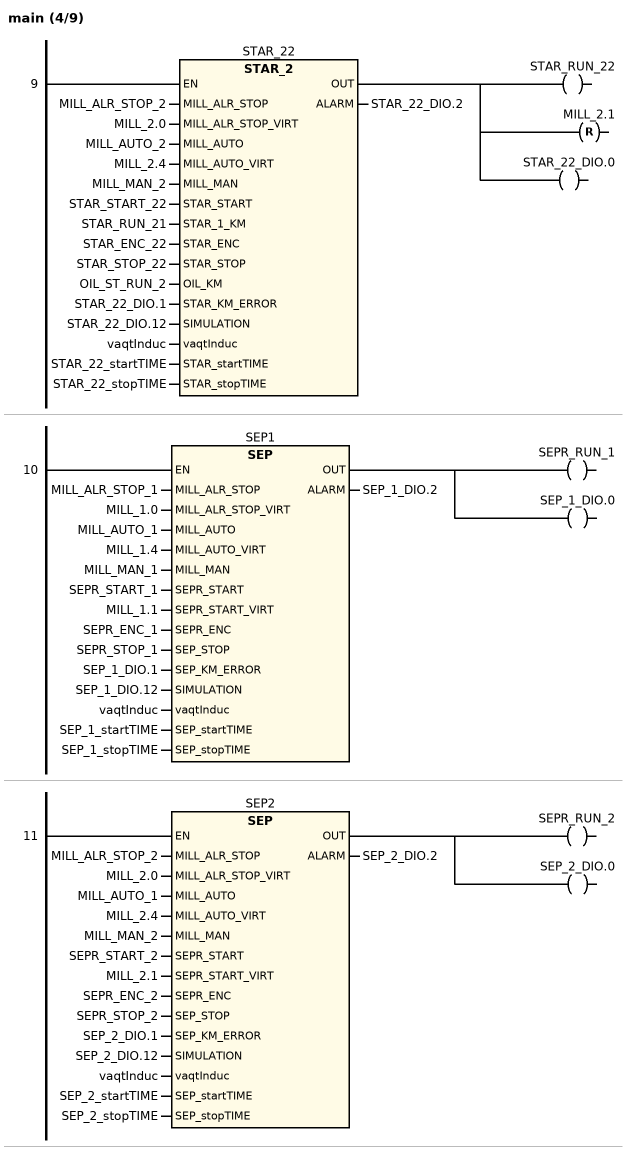
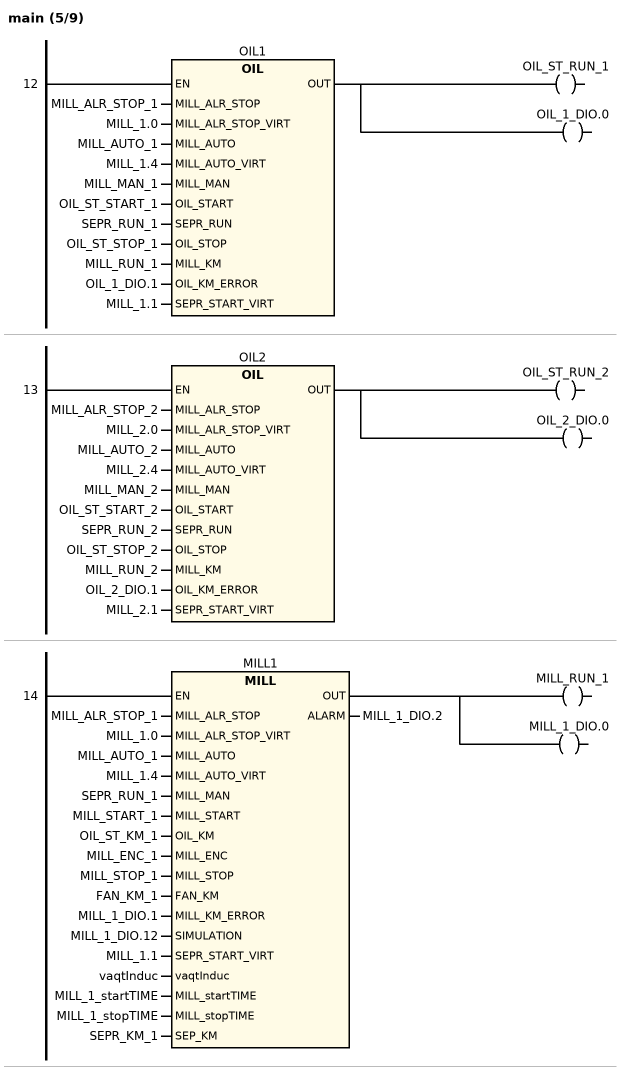
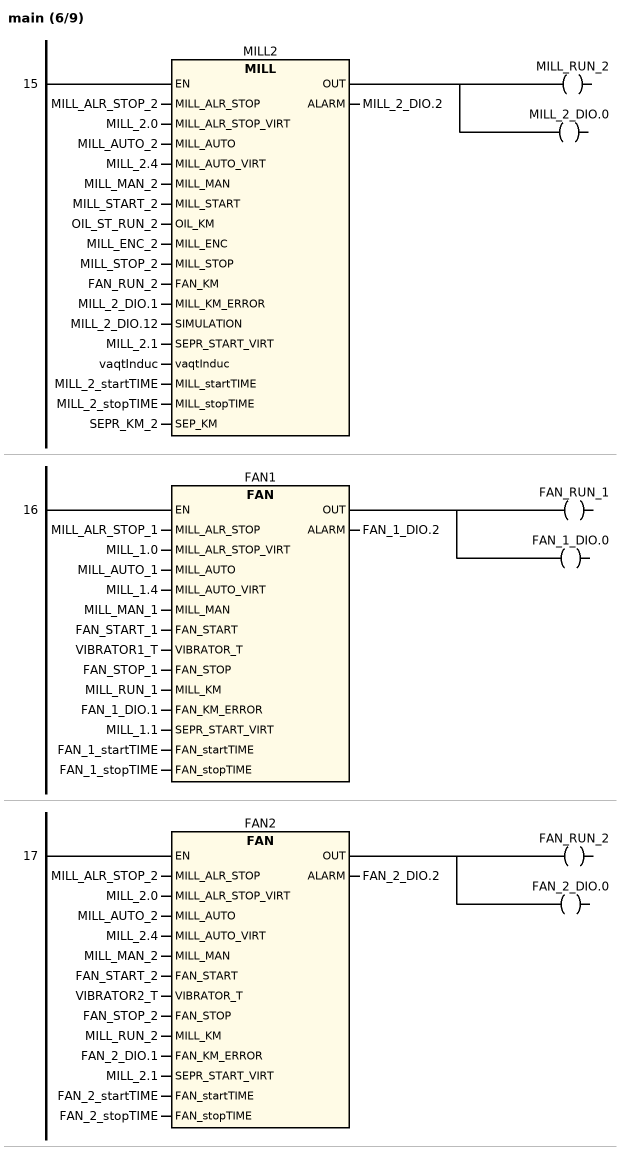
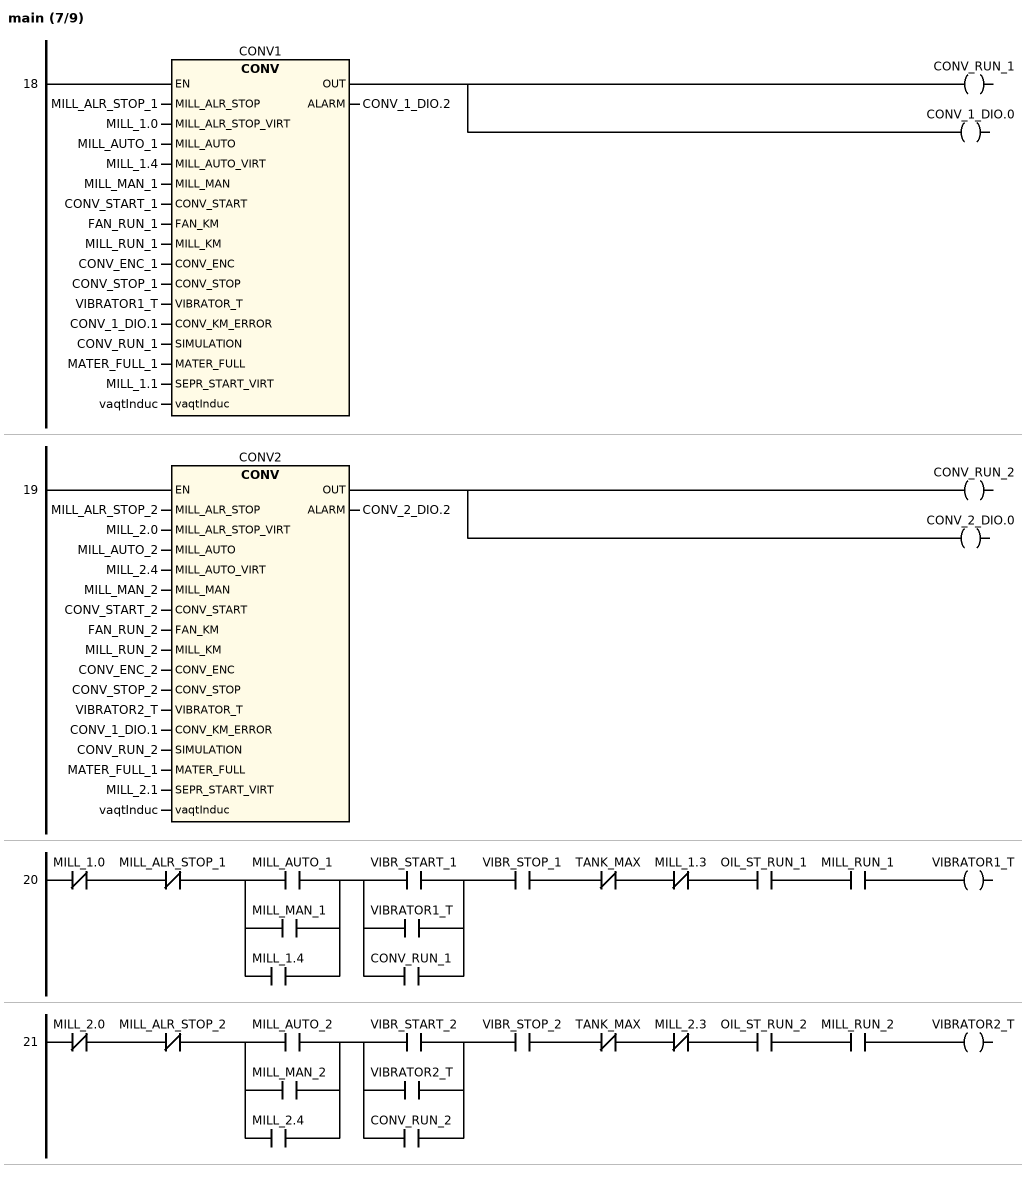
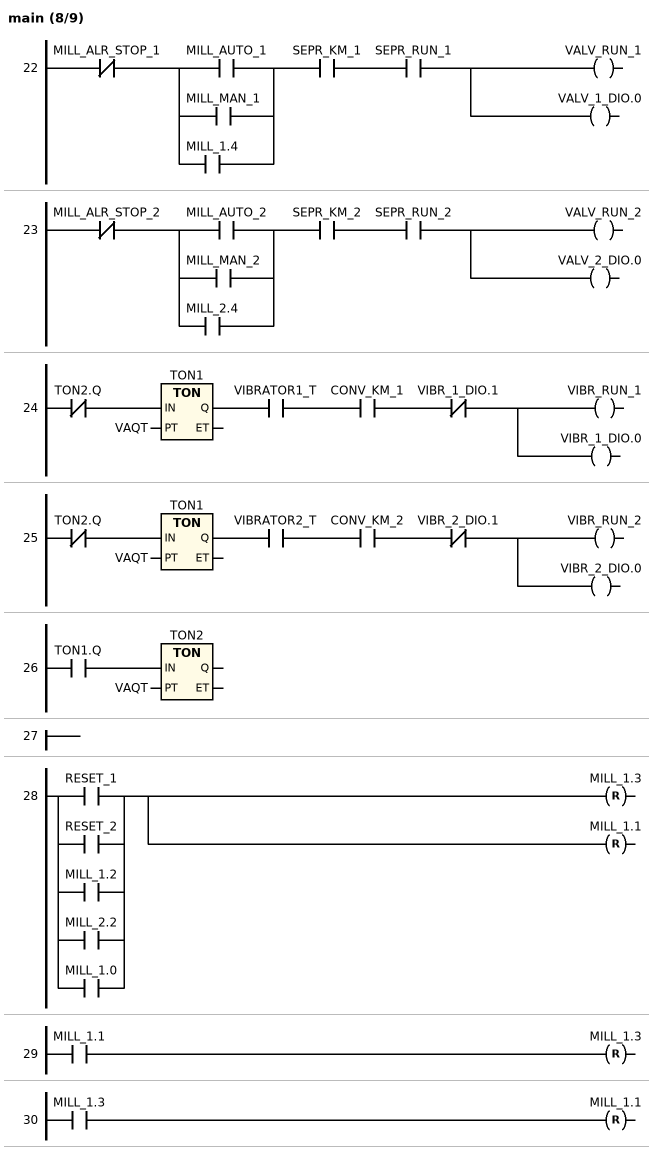
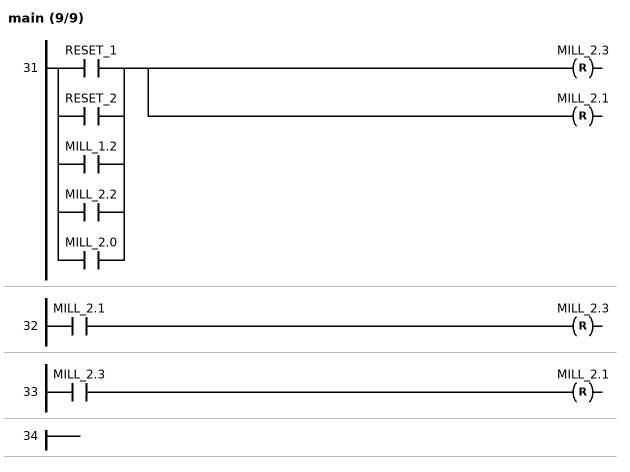
_LD_ (* Ladder Diagram *)
NETWORK 1
	EL_12:ELEV(EN: *, MILL_ALR_STOP1: MILL_ALR_STOP_1, MILL_ALR_STOP2: MILL_ALR_STOP_2, MILL_ALR_STOP_VIRT1: MILL_1.0, MILL_ALR_STOP_VIRT2: MILL_2.0, MILL_AUTO1: MILL_AUTO_1, MILL_AUTO2: MILL_AUTO_2, MILL_AUTO_VIRT1: MILL_1.4, MILL_AUTO_VIRT2: MILL_2.4, TANK_MAX: TANK_MAX, MILL_MAN1: MILL_MAN_1, MILL_MAN2: MILL_MAN_2, ELEV_START1: ELV_START_1, ELEV_START2: ELV_START_2, VIBR_RUN_1: VIBRATOR1_T, VIBR_RUN_2: VIBRATOR2_T, ELEV_ENC: ELV_ENC_2, ELEV_STOP1: ELV_STOP_1, ELEV_STOP2: ELV_STOP_2, SHNK_KM1: SHNK_KM_1, SHNK_KM2: SHNK_KM_2, ELEV_KM_ERROR: ELEV_12_DIO.1, SIMULATION: ELEV_12_DIO.12, SEPR_START_VIRT1: MILL_1.1, SEPR_START_VIRT2: MILL_2.1, vaqtInduc: vaqtInduc, ELEV_startTIME: ELEV_12_startTIME, ELEV_stopTIME: ELEV_12_stopTIME, ALARM => ELEV_12_DIO.2) --- (ELV_RUN) (ELEV_12_DIO.0)
NETWORK 2
	SHNK1:SHNEK(EN: *, MILL_ALR_STOP: MILL_ALR_STOP_1, MILL_ALR_STOP_VIRT: MILL_1.0, MILL_AUTO: MILL_AUTO_1, MILL_AUTO_VIRT: MILL_1.4, MILL_MAN: MILL_MAN_1, SHNK_START: SHNK_START_1, SEP_RUN: SEPR_RUN_1, ELEV_KM: ELV_RUN, SHNK_ENC: SHNK_ENC_1, SHNK_STOP: SHNK_STOP_1, SHNK_SIKL_KM: SHNK_SKL_RUN_1, SHNK_KM_ERROR: SHNEK_1_DIO.1, SIMULATION: SHNEK_1_DIO.12, SEPR_START_VIRT: MILL_1.1, vaqtInduc: vaqtInduc, SHNK_startTIME: SHNEK_1_startTIME, SHNK_stopTIME: SHNEK_1_stopTIME, ALARM => SHNEK_1_DIO.2) --- (SHNK_RUN_1) (SHNEK_1_DIO.0)
NETWORK 3
	SHNK2:SHNEK(EN: *, MILL_ALR_STOP: MILL_ALR_STOP_2, MILL_ALR_STOP_VIRT: MILL_2.0, MILL_AUTO: MILL_AUTO_2, MILL_AUTO_VIRT: MILL_2.4, MILL_MAN: MILL_MAN_2, SHNK_START: SHNK_START_2, SEP_RUN: SEPR_RUN_2, ELEV_KM: ELV_RUN, SHNK_ENC: SHNK_ENC_2, SHNK_STOP: SHNK_STOP_2, SHNK_SIKL_KM: SHNK_SKL_RUN_2, SHNK_KM_ERROR: SHNEK_2_DIO.1, SIMULATION: SHNEK_2_DIO.12, SEPR_START_VIRT: MILL_2.1, vaqtInduc: vaqtInduc, SHNK_startTIME: SHNEK_2_startTIME, SHNK_stopTIME: SHNEK_2_stopTIME, ALARM => SHNEK_2_DIO.2) --- (SHNK_RUN_2) (SHNEK_2_DIO.0)
NETWORK 4
	SHNEK_SIKL1:SHNEK_SIKL(EN: *, MILL_ALR_STOP: MILL_ALR_STOP_1, MILL_ALR_STOP_VIRT: MILL_1.0, MILL_AUTO: MILL_AUTO_1, MILL_AUTO_VIRT: MILL_1.4, MILL_MAN: MILL_MAN_1, SHNK_SIKL_START: SHNK_SKL_START_1, SHNK_KM: SHNK_RUN_1, SHNK_SIKL_ENC: SHNK_SKL_ENC_1, SHNK_SIKL_STOP: SHNK_SKL_STOP_1, STAR_1_KM: STAR_RUN_11, SHNK_SIKL_KM_ERROR: SHNK_SIKL_1_DIO.1, SIMULATION: SHNK_SIKL_1_DIO.12, SEPR_START_VIRT: MILL_1.1, vaqtInduc: vaqtInduc, SHNK_SIKL_startTIME: SHNK_SIKL_1_startTIME, SHNK_SIKL_stopTIME: SHNK_SIKL_1_stopTIME, ALARM => SHNK_SIKL_1_DIO.2) --- (SHNK_SKL_RUN_1) (SHNK_SIKL_1_DIO.0)
NETWORK 5
	SHNEK_SIKL2:SHNEK_SIKL(EN: *, MILL_ALR_STOP: MILL_ALR_STOP_2, MILL_ALR_STOP_VIRT: MILL_2.0, MILL_AUTO: MILL_AUTO_2, MILL_AUTO_VIRT: MILL_2.4, MILL_MAN: MILL_MAN_2, SHNK_SIKL_START: SHNK_SKL_START_2, SHNK_KM: SHNK_RUN_2, SHNK_SIKL_ENC: SHNK_SKL_ENC_2, SHNK_SIKL_STOP: SHNK_SKL_STOP_2, STAR_1_KM: STAR_RUN_21, SHNK_SIKL_KM_ERROR: SHNK_SIKL_2_DIO.1, SIMULATION: SHNK_SIKL_2_DIO.12, SEPR_START_VIRT: MILL_2.1, vaqtInduc: vaqtInduc, SHNK_SIKL_startTIME: SHNK_SIKL_2_startTIME, SHNK_SIKL_stopTIME: SHNK_SIKL_2_stopTIME, ALARM => SHNK_SIKL_2_DIO.2) --- (SHNK_SKL_RUN_2) (SHNK_SIKL_2_DIO.0)
NETWORK 6
	STAR_11:STAR_1(EN: *, MILL_ALR_STOP: MILL_ALR_STOP_1, MILL_ALR_STOP_VIRT: MILL_1.0, MILL_AUTO: MILL_AUTO_1, MILL_AUTO_VIRT: MILL_1.4, MILL_MAN: MILL_MAN_1, STAR_START: STAR_START_11, SHNK_SIKL_KM: SHNK_SKL_RUN_1, STAR_ENC: STAR_ENC_11, STAR_STOP: STAR_STOP_11, STAR_2_KM: STAR_RUN_12, STAR_KM_ERROR: STAR_11_DIO.1, SIMULATION: STAR_11_DIO.12, SEPR_START_VIRT: MILL_1.1, vaqtInduc: vaqtInduc, STAR_startTIME: STAR_11_startTIME, STAR_stopTIME: STAR_11_stopTIME, ALARM => STAR_11_DIO.2) --- (STAR_RUN_11) (STAR_11_DIO.0)
NETWORK 7
	STAR_21:STAR_1(EN: *, MILL_ALR_STOP: MILL_ALR_STOP_2, MILL_ALR_STOP_VIRT: MILL_2.0, MILL_AUTO: MILL_AUTO_2, MILL_AUTO_VIRT: MILL_2.4, MILL_MAN: MILL_MAN_2, STAR_START: STAR_START_21, SHNK_SIKL_KM: SHNK_SKL_RUN_2, STAR_ENC: STAR_ENC_21, STAR_STOP: STAR_STOP_21, STAR_2_KM: STAR_RUN_22, STAR_KM_ERROR: STAR_21_DIO.1, SIMULATION: STAR_21_DIO.12, SEPR_START_VIRT: MILL_2.1, vaqtInduc: vaqtInduc, STAR_startTIME: STAR_21_startTIME, STAR_stopTIME: STAR_21_stopTIME, ALARM => STAR_21_DIO.2) --- (STAR_RUN_21) (STAR_21_DIO.0)
NETWORK 8
	STAR_12:STAR_2(EN: *, MILL_ALR_STOP: MILL_ALR_STOP_1, MILL_ALR_STOP_VIRT: MILL_1.0, MILL_AUTO: MILL_AUTO_1, MILL_AUTO_VIRT: MILL_1.4, MILL_MAN: MILL_MAN_1, STAR_START: STAR_START_12, STAR_1_KM: STAR_RUN_11, STAR_ENC: STAR_ENC_12, STAR_STOP: STAR_STOP_12, OIL_KM: OIL_ST_RUN_1, STAR_KM_ERROR: STAR_12_DIO.1, SIMULATION: STAR_12_DIO.12, vaqtInduc: vaqtInduc, STAR_startTIME: STAR_12_startTIME, STAR_stopTIME: STAR_12_stopTIME, ALARM => STAR_12_DIO.2) --- (STAR_RUN_12) (R MILL_1.1) (STAR_12_DIO.0)
NETWORK 9
	STAR_22:STAR_2(EN: *, MILL_ALR_STOP: MILL_ALR_STOP_2, MILL_ALR_STOP_VIRT: MILL_2.0, MILL_AUTO: MILL_AUTO_2, MILL_AUTO_VIRT: MILL_2.4, MILL_MAN: MILL_MAN_2, STAR_START: STAR_START_22, STAR_1_KM: STAR_RUN_21, STAR_ENC: STAR_ENC_22, STAR_STOP: STAR_STOP_22, OIL_KM: OIL_ST_RUN_2, STAR_KM_ERROR: STAR_22_DIO.1, SIMULATION: STAR_22_DIO.12, vaqtInduc: vaqtInduc, STAR_startTIME: STAR_22_startTIME, STAR_stopTIME: STAR_22_stopTIME, ALARM => STAR_22_DIO.2) --- (STAR_RUN_22) (R MILL_2.1) (STAR_22_DIO.0)
NETWORK 10
	SEP1:SEP(EN: *, MILL_ALR_STOP: MILL_ALR_STOP_1, MILL_ALR_STOP_VIRT: MILL_1.0, MILL_AUTO: MILL_AUTO_1, MILL_AUTO_VIRT: MILL_1.4, MILL_MAN: MILL_MAN_1, SEPR_START: SEPR_START_1, SEPR_START_VIRT: MILL_1.1, SEPR_ENC: SEPR_ENC_1, SEP_STOP: SEPR_STOP_1, SEP_KM_ERROR: SEP_1_DIO.1, SIMULATION: SEP_1_DIO.12, vaqtInduc: vaqtInduc, SEP_startTIME: SEP_1_startTIME, SEP_stopTIME: SEP_1_stopTIME, ALARM => SEP_1_DIO.2) --- (SEPR_RUN_1) (SEP_1_DIO.0)
NETWORK 11
	SEP2:SEP(EN: *, MILL_ALR_STOP: MILL_ALR_STOP_2, MILL_ALR_STOP_VIRT: MILL_2.0, MILL_AUTO: MILL_AUTO_1, MILL_AUTO_VIRT: MILL_2.4, MILL_MAN: MILL_MAN_2, SEPR_START: SEPR_START_2, SEPR_START_VIRT: MILL_2.1, SEPR_ENC: SEPR_ENC_2, SEP_STOP: SEPR_STOP_2, SEP_KM_ERROR: SEP_2_DIO.1, SIMULATION: SEP_2_DIO.12, vaqtInduc: vaqtInduc, SEP_startTIME: SEP_2_startTIME, SEP_stopTIME: SEP_2_stopTIME, ALARM => SEP_2_DIO.2) --- (SEPR_RUN_2) (SEP_2_DIO.0)
NETWORK 12
	OIL1:OIL(EN: *, MILL_ALR_STOP: MILL_ALR_STOP_1, MILL_ALR_STOP_VIRT: MILL_1.0, MILL_AUTO: MILL_AUTO_1, MILL_AUTO_VIRT: MILL_1.4, MILL_MAN: MILL_MAN_1, OIL_START: OIL_ST_START_1, SEPR_RUN: SEPR_RUN_1, OIL_STOP: OIL_ST_STOP_1, MILL_KM: MILL_RUN_1, OIL_KM_ERROR: OIL_1_DIO.1, SEPR_START_VIRT: MILL_1.1) --- (OIL_ST_RUN_1) (OIL_1_DIO.0)
NETWORK 13
	OIL2:OIL(EN: *, MILL_ALR_STOP: MILL_ALR_STOP_2, MILL_ALR_STOP_VIRT: MILL_2.0, MILL_AUTO: MILL_AUTO_2, MILL_AUTO_VIRT: MILL_2.4, MILL_MAN: MILL_MAN_2, OIL_START: OIL_ST_START_2, SEPR_RUN: SEPR_RUN_2, OIL_STOP: OIL_ST_STOP_2, MILL_KM: MILL_RUN_2, OIL_KM_ERROR: OIL_2_DIO.1, SEPR_START_VIRT: MILL_2.1) --- (OIL_ST_RUN_2) (OIL_2_DIO.0)
NETWORK 14
	MILL1:MILL(EN: *, MILL_ALR_STOP: MILL_ALR_STOP_1, MILL_ALR_STOP_VIRT: MILL_1.0, MILL_AUTO: MILL_AUTO_1, MILL_AUTO_VIRT: MILL_1.4, MILL_MAN: SEPR_RUN_1, MILL_START: MILL_START_1, OIL_KM: OIL_ST_KM_1, MILL_ENC: MILL_ENC_1, MILL_STOP: MILL_STOP_1, FAN_KM: FAN_KM_1, MILL_KM_ERROR: MILL_1_DIO.1, SIMULATION: MILL_1_DIO.12, SEPR_START_VIRT: MILL_1.1, vaqtInduc: vaqtInduc, MILL_startTIME: MILL_1_startTIME, MILL_stopTIME: MILL_1_stopTIME, SEP_KM: SEPR_KM_1, ALARM => MILL_1_DIO.2) --- (MILL_RUN_1) (MILL_1_DIO.0)
NETWORK 15
	MILL2:MILL(EN: *, MILL_ALR_STOP: MILL_ALR_STOP_2, MILL_ALR_STOP_VIRT: MILL_2.0, MILL_AUTO: MILL_AUTO_2, MILL_AUTO_VIRT: MILL_2.4, MILL_MAN: MILL_MAN_2, MILL_START: MILL_START_2, OIL_KM: OIL_ST_RUN_2, MILL_ENC: MILL_ENC_2, MILL_STOP: MILL_STOP_2, FAN_KM: FAN_RUN_2, MILL_KM_ERROR: MILL_2_DIO.1, SIMULATION: MILL_2_DIO.12, SEPR_START_VIRT: MILL_2.1, vaqtInduc: vaqtInduc, MILL_startTIME: MILL_2_startTIME, MILL_stopTIME: MILL_2_stopTIME, SEP_KM: SEPR_KM_2, ALARM => MILL_2_DIO.2) --- (MILL_RUN_2) (MILL_2_DIO.0)
NETWORK 16
	FAN1:FAN(EN: *, MILL_ALR_STOP: MILL_ALR_STOP_1, MILL_ALR_STOP_VIRT: MILL_1.0, MILL_AUTO: MILL_AUTO_1, MILL_AUTO_VIRT: MILL_1.4, MILL_MAN: MILL_MAN_1, FAN_START: FAN_START_1, VIBRATOR_T: VIBRATOR1_T, FAN_STOP: FAN_STOP_1, MILL_KM: MILL_RUN_1, FAN_KM_ERROR: FAN_1_DIO.1, SEPR_START_VIRT: MILL_1.1, FAN_startTIME: FAN_1_startTIME, FAN_stopTIME: FAN_1_stopTIME, ALARM => FAN_1_DIO.2) --- (FAN_RUN_1) (FAN_1_DIO.0)
NETWORK 17
	FAN2:FAN(EN: *, MILL_ALR_STOP: MILL_ALR_STOP_2, MILL_ALR_STOP_VIRT: MILL_2.0, MILL_AUTO: MILL_AUTO_2, MILL_AUTO_VIRT: MILL_2.4, MILL_MAN: MILL_MAN_2, FAN_START: FAN_START_2, VIBRATOR_T: VIBRATOR2_T, FAN_STOP: FAN_STOP_2, MILL_KM: MILL_RUN_2, FAN_KM_ERROR: FAN_2_DIO.1, SEPR_START_VIRT: MILL_2.1, FAN_startTIME: FAN_2_startTIME, FAN_stopTIME: FAN_2_stopTIME, ALARM => FAN_2_DIO.2) --- (FAN_RUN_2) (FAN_2_DIO.0)
NETWORK 18
	CONV1:CONV(EN: *, MILL_ALR_STOP: MILL_ALR_STOP_1, MILL_ALR_STOP_VIRT: MILL_1.0, MILL_AUTO: MILL_AUTO_1, MILL_AUTO_VIRT: MILL_1.4, MILL_MAN: MILL_MAN_1, CONV_START: CONV_START_1, FAN_KM: FAN_RUN_1, MILL_KM: MILL_RUN_1, CONV_ENC: CONV_ENC_1, CONV_STOP: CONV_STOP_1, VIBRATOR_T: VIBRATOR1_T, CONV_KM_ERROR: CONV_1_DIO.1, SIMULATION: CONV_RUN_1, MATER_FULL: MATER_FULL_1, SEPR_START_VIRT: MILL_1.1, vaqtInduc: vaqtInduc, ALARM => CONV_1_DIO.2) --- (CONV_RUN_1) (CONV_1_DIO.0)
NETWORK 19
	CONV2:CONV(EN: *, MILL_ALR_STOP: MILL_ALR_STOP_2, MILL_ALR_STOP_VIRT: MILL_2.0, MILL_AUTO: MILL_AUTO_2, MILL_AUTO_VIRT: MILL_2.4, MILL_MAN: MILL_MAN_2, CONV_START: CONV_START_2, FAN_KM: FAN_RUN_2, MILL_KM: MILL_RUN_2, CONV_ENC: CONV_ENC_2, CONV_STOP: CONV_STOP_2, VIBRATOR_T: VIBRATOR2_T, CONV_KM_ERROR: CONV_1_DIO.1, SIMULATION: CONV_RUN_2, MATER_FULL: MATER_FULL_1, SEPR_START_VIRT: MILL_2.1, vaqtInduc: vaqtInduc, ALARM => CONV_2_DIO.2) --- (CONV_RUN_2) (CONV_2_DIO.0)
NETWORK 20
	[/MILL_1.0] - [/MILL_ALR_STOP_1] - { [MILL_AUTO_1] | [MILL_MAN_1] | [MILL_1.4] } - { [VIBR_START_1] | [VIBRATOR1_T] | [CONV_RUN_1] } - [VIBR_STOP_1] - [/TANK_MAX] - [/MILL_1.3] - [OIL_ST_RUN_1] - [MILL_RUN_1] --- (VIBRATOR1_T)
NETWORK 21
	[/MILL_2.0] - [/MILL_ALR_STOP_2] - { [MILL_AUTO_2] | [MILL_MAN_2] | [MILL_2.4] } - { [VIBR_START_2] | [VIBRATOR2_T] | [CONV_RUN_2] } - [VIBR_STOP_2] - [/TANK_MAX] - [/MILL_2.3] - [OIL_ST_RUN_2] - [MILL_RUN_2] --- (VIBRATOR2_T)
NETWORK 22
	[/MILL_ALR_STOP_1] - { [MILL_AUTO_1] | [MILL_MAN_1] | [MILL_1.4] } - [SEPR_KM_1] - [SEPR_RUN_1] --- (VALV_RUN_1) (VALV_1_DIO.0)
NETWORK 23
	[/MILL_ALR_STOP_2] - { [MILL_AUTO_2] | [MILL_MAN_2] | [MILL_2.4] } - [SEPR_KM_2] - [SEPR_RUN_2] --- (VALV_RUN_2) (VALV_2_DIO.0)
NETWORK 24
	[/TON2.Q] - TON1:TON(IN: *, PT: VAQT) - [VIBRATOR1_T] - [CONV_KM_1] - [/VIBR_1_DIO.1] --- (VIBR_RUN_1) (VIBR_1_DIO.0)
NETWORK 25
	[/TON2.Q] - TON1:TON(IN: *, PT: VAQT) - [VIBRATOR2_T] - [CONV_KM_2] - [/VIBR_2_DIO.1] --- (VIBR_RUN_2) (VIBR_2_DIO.0)
NETWORK 26
	[TON1.Q] - TON2:TON(IN: *, PT: VAQT)
NETWORK 27
	*
NETWORK 28
	{ [RESET_1] | [RESET_2] | [MILL_1.2] | [MILL_2.2] | [MILL_1.0] } --- (R MILL_1.3) (R MILL_1.1)
NETWORK 29
	[MILL_1.1] --- (R MILL_1.3)
NETWORK 30
	[MILL_1.3] --- (R MILL_1.1)
NETWORK 31
	{ [RESET_1] | [RESET_2] | [MILL_1.2] | [MILL_2.2] | [MILL_2.0] } --- (R MILL_2.3) (R MILL_2.1)
NETWORK 32
	[MILL_2.1] --- (R MILL_2.3)
NETWORK 33
	[MILL_2.3] --- (R MILL_2.1)
NETWORK 34
	*
_END_LD_
(* the same logic as Structured Text *)
(* Network 1 *)
EL_12(EN := TRUE, MILL_ALR_STOP1 := MILL_ALR_STOP_1, MILL_ALR_STOP2 := MILL_ALR_STOP_2, MILL_ALR_STOP_VIRT1 := MILL_1.0, MILL_ALR_STOP_VIRT2 := MILL_2.0, MILL_AUTO1 := MILL_AUTO_1, MILL_AUTO2 := MILL_AUTO_2, MILL_AUTO_VIRT1 := MILL_1.4, MILL_AUTO_VIRT2 := MILL_2.4, TANK_MAX := TANK_MAX, MILL_MAN1 := MILL_MAN_1, MILL_MAN2 := MILL_MAN_2, ELEV_START1 := ELV_START_1, ELEV_START2 := ELV_START_2, VIBR_RUN_1 := VIBRATOR1_T, VIBR_RUN_2 := VIBRATOR2_T, ELEV_ENC := ELV_ENC_2, ELEV_STOP1 := ELV_STOP_1, ELEV_STOP2 := ELV_STOP_2, SHNK_KM1 := SHNK_KM_1, SHNK_KM2 := SHNK_KM_2, ELEV_KM_ERROR := ELEV_12_DIO.1, SIMULATION := ELEV_12_DIO.12, SEPR_START_VIRT1 := MILL_1.1, SEPR_START_VIRT2 := MILL_2.1, vaqtInduc := vaqtInduc, ELEV_startTIME := ELEV_12_startTIME, ELEV_stopTIME := ELEV_12_stopTIME);
ELEV_12_DIO.2 := EL_12.ALARM;
ELV_RUN := EL_12.OUT;
ELEV_12_DIO.0 := EL_12.OUT;
(* Network 2 *)
SHNK1(EN := TRUE, MILL_ALR_STOP := MILL_ALR_STOP_1, MILL_ALR_STOP_VIRT := MILL_1.0, MILL_AUTO := MILL_AUTO_1, MILL_AUTO_VIRT := MILL_1.4, MILL_MAN := MILL_MAN_1, SHNK_START := SHNK_START_1, SEP_RUN := SEPR_RUN_1, ELEV_KM := ELV_RUN, SHNK_ENC := SHNK_ENC_1, SHNK_STOP := SHNK_STOP_1, SHNK_SIKL_KM := SHNK_SKL_RUN_1, SHNK_KM_ERROR := SHNEK_1_DIO.1, SIMULATION := SHNEK_1_DIO.12, SEPR_START_VIRT := MILL_1.1, vaqtInduc := vaqtInduc, SHNK_startTIME := SHNEK_1_startTIME, SHNK_stopTIME := SHNEK_1_stopTIME);
SHNEK_1_DIO.2 := SHNK1.ALARM;
SHNK_RUN_1 := SHNK1.OUT;
SHNEK_1_DIO.0 := SHNK1.OUT;
(* Network 3 *)
SHNK2(EN := TRUE, MILL_ALR_STOP := MILL_ALR_STOP_2, MILL_ALR_STOP_VIRT := MILL_2.0, MILL_AUTO := MILL_AUTO_2, MILL_AUTO_VIRT := MILL_2.4, MILL_MAN := MILL_MAN_2, SHNK_START := SHNK_START_2, SEP_RUN := SEPR_RUN_2, ELEV_KM := ELV_RUN, SHNK_ENC := SHNK_ENC_2, SHNK_STOP := SHNK_STOP_2, SHNK_SIKL_KM := SHNK_SKL_RUN_2, SHNK_KM_ERROR := SHNEK_2_DIO.1, SIMULATION := SHNEK_2_DIO.12, SEPR_START_VIRT := MILL_2.1, vaqtInduc := vaqtInduc, SHNK_startTIME := SHNEK_2_startTIME, SHNK_stopTIME := SHNEK_2_stopTIME);
SHNEK_2_DIO.2 := SHNK2.ALARM;
SHNK_RUN_2 := SHNK2.OUT;
SHNEK_2_DIO.0 := SHNK2.OUT;
(* Network 4 *)
SHNEK_SIKL1(EN := TRUE, MILL_ALR_STOP := MILL_ALR_STOP_1, MILL_ALR_STOP_VIRT := MILL_1.0, MILL_AUTO := MILL_AUTO_1, MILL_AUTO_VIRT := MILL_1.4, MILL_MAN := MILL_MAN_1, SHNK_SIKL_START := SHNK_SKL_START_1, SHNK_KM := SHNK_RUN_1, SHNK_SIKL_ENC := SHNK_SKL_ENC_1, SHNK_SIKL_STOP := SHNK_SKL_STOP_1, STAR_1_KM := STAR_RUN_11, SHNK_SIKL_KM_ERROR := SHNK_SIKL_1_DIO.1, SIMULATION := SHNK_SIKL_1_DIO.12, SEPR_START_VIRT := MILL_1.1, vaqtInduc := vaqtInduc, SHNK_SIKL_startTIME := SHNK_SIKL_1_startTIME, SHNK_SIKL_stopTIME := SHNK_SIKL_1_stopTIME);
SHNK_SIKL_1_DIO.2 := SHNEK_SIKL1.ALARM;
SHNK_SKL_RUN_1 := SHNEK_SIKL1.OUT;
SHNK_SIKL_1_DIO.0 := SHNEK_SIKL1.OUT;
(* Network 5 *)
SHNEK_SIKL2(EN := TRUE, MILL_ALR_STOP := MILL_ALR_STOP_2, MILL_ALR_STOP_VIRT := MILL_2.0, MILL_AUTO := MILL_AUTO_2, MILL_AUTO_VIRT := MILL_2.4, MILL_MAN := MILL_MAN_2, SHNK_SIKL_START := SHNK_SKL_START_2, SHNK_KM := SHNK_RUN_2, SHNK_SIKL_ENC := SHNK_SKL_ENC_2, SHNK_SIKL_STOP := SHNK_SKL_STOP_2, STAR_1_KM := STAR_RUN_21, SHNK_SIKL_KM_ERROR := SHNK_SIKL_2_DIO.1, SIMULATION := SHNK_SIKL_2_DIO.12, SEPR_START_VIRT := MILL_2.1, vaqtInduc := vaqtInduc, SHNK_SIKL_startTIME := SHNK_SIKL_2_startTIME, SHNK_SIKL_stopTIME := SHNK_SIKL_2_stopTIME);
SHNK_SIKL_2_DIO.2 := SHNEK_SIKL2.ALARM;
SHNK_SKL_RUN_2 := SHNEK_SIKL2.OUT;
SHNK_SIKL_2_DIO.0 := SHNEK_SIKL2.OUT;
(* Network 6 *)
STAR_11(EN := TRUE, MILL_ALR_STOP := MILL_ALR_STOP_1, MILL_ALR_STOP_VIRT := MILL_1.0, MILL_AUTO := MILL_AUTO_1, MILL_AUTO_VIRT := MILL_1.4, MILL_MAN := MILL_MAN_1, STAR_START := STAR_START_11, SHNK_SIKL_KM := SHNK_SKL_RUN_1, STAR_ENC := STAR_ENC_11, STAR_STOP := STAR_STOP_11, STAR_2_KM := STAR_RUN_12, STAR_KM_ERROR := STAR_11_DIO.1, SIMULATION := STAR_11_DIO.12, SEPR_START_VIRT := MILL_1.1, vaqtInduc := vaqtInduc, STAR_startTIME := STAR_11_startTIME, STAR_stopTIME := STAR_11_stopTIME);
STAR_11_DIO.2 := STAR_11.ALARM;
STAR_RUN_11 := STAR_11.OUT;
STAR_11_DIO.0 := STAR_11.OUT;
(* Network 7 *)
STAR_21(EN := TRUE, MILL_ALR_STOP := MILL_ALR_STOP_2, MILL_ALR_STOP_VIRT := MILL_2.0, MILL_AUTO := MILL_AUTO_2, MILL_AUTO_VIRT := MILL_2.4, MILL_MAN := MILL_MAN_2, STAR_START := STAR_START_21, SHNK_SIKL_KM := SHNK_SKL_RUN_2, STAR_ENC := STAR_ENC_21, STAR_STOP := STAR_STOP_21, STAR_2_KM := STAR_RUN_22, STAR_KM_ERROR := STAR_21_DIO.1, SIMULATION := STAR_21_DIO.12, SEPR_START_VIRT := MILL_2.1, vaqtInduc := vaqtInduc, STAR_startTIME := STAR_21_startTIME, STAR_stopTIME := STAR_21_stopTIME);
STAR_21_DIO.2 := STAR_21.ALARM;
STAR_RUN_21 := STAR_21.OUT;
STAR_21_DIO.0 := STAR_21.OUT;
(* Network 8 *)
STAR_12(EN := TRUE, MILL_ALR_STOP := MILL_ALR_STOP_1, MILL_ALR_STOP_VIRT := MILL_1.0, MILL_AUTO := MILL_AUTO_1, MILL_AUTO_VIRT := MILL_1.4, MILL_MAN := MILL_MAN_1, STAR_START := STAR_START_12, STAR_1_KM := STAR_RUN_11, STAR_ENC := STAR_ENC_12, STAR_STOP := STAR_STOP_12, OIL_KM := OIL_ST_RUN_1, STAR_KM_ERROR := STAR_12_DIO.1, SIMULATION := STAR_12_DIO.12, vaqtInduc := vaqtInduc, STAR_startTIME := STAR_12_startTIME, STAR_stopTIME := STAR_12_stopTIME);
STAR_12_DIO.2 := STAR_12.ALARM;
STAR_RUN_12 := STAR_12.OUT;
IF STAR_12.OUT THEN MILL_1.1 := FALSE; END_IF;
STAR_12_DIO.0 := STAR_12.OUT;
(* Network 9 *)
STAR_22(EN := TRUE, MILL_ALR_STOP := MILL_ALR_STOP_2, MILL_ALR_STOP_VIRT := MILL_2.0, MILL_AUTO := MILL_AUTO_2, MILL_AUTO_VIRT := MILL_2.4, MILL_MAN := MILL_MAN_2, STAR_START := STAR_START_22, STAR_1_KM := STAR_RUN_21, STAR_ENC := STAR_ENC_22, STAR_STOP := STAR_STOP_22, OIL_KM := OIL_ST_RUN_2, STAR_KM_ERROR := STAR_22_DIO.1, SIMULATION := STAR_22_DIO.12, vaqtInduc := vaqtInduc, STAR_startTIME := STAR_22_startTIME, STAR_stopTIME := STAR_22_stopTIME);
STAR_22_DIO.2 := STAR_22.ALARM;
STAR_RUN_22 := STAR_22.OUT;
IF STAR_22.OUT THEN MILL_2.1 := FALSE; END_IF;
STAR_22_DIO.0 := STAR_22.OUT;
(* Network 10 *)
SEP1(EN := TRUE, MILL_ALR_STOP := MILL_ALR_STOP_1, MILL_ALR_STOP_VIRT := MILL_1.0, MILL_AUTO := MILL_AUTO_1, MILL_AUTO_VIRT := MILL_1.4, MILL_MAN := MILL_MAN_1, SEPR_START := SEPR_START_1, SEPR_START_VIRT := MILL_1.1, SEPR_ENC := SEPR_ENC_1, SEP_STOP := SEPR_STOP_1, SEP_KM_ERROR := SEP_1_DIO.1, SIMULATION := SEP_1_DIO.12, vaqtInduc := vaqtInduc, SEP_startTIME := SEP_1_startTIME, SEP_stopTIME := SEP_1_stopTIME);
SEP_1_DIO.2 := SEP1.ALARM;
SEPR_RUN_1 := SEP1.OUT;
SEP_1_DIO.0 := SEP1.OUT;
(* Network 11 *)
SEP2(EN := TRUE, MILL_ALR_STOP := MILL_ALR_STOP_2, MILL_ALR_STOP_VIRT := MILL_2.0, MILL_AUTO := MILL_AUTO_1, MILL_AUTO_VIRT := MILL_2.4, MILL_MAN := MILL_MAN_2, SEPR_START := SEPR_START_2, SEPR_START_VIRT := MILL_2.1, SEPR_ENC := SEPR_ENC_2, SEP_STOP := SEPR_STOP_2, SEP_KM_ERROR := SEP_2_DIO.1, SIMULATION := SEP_2_DIO.12, vaqtInduc := vaqtInduc, SEP_startTIME := SEP_2_startTIME, SEP_stopTIME := SEP_2_stopTIME);
SEP_2_DIO.2 := SEP2.ALARM;
SEPR_RUN_2 := SEP2.OUT;
SEP_2_DIO.0 := SEP2.OUT;
(* Network 12 *)
OIL1(EN := TRUE, MILL_ALR_STOP := MILL_ALR_STOP_1, MILL_ALR_STOP_VIRT := MILL_1.0, MILL_AUTO := MILL_AUTO_1, MILL_AUTO_VIRT := MILL_1.4, MILL_MAN := MILL_MAN_1, OIL_START := OIL_ST_START_1, SEPR_RUN := SEPR_RUN_1, OIL_STOP := OIL_ST_STOP_1, MILL_KM := MILL_RUN_1, OIL_KM_ERROR := OIL_1_DIO.1, SEPR_START_VIRT := MILL_1.1);
OIL_ST_RUN_1 := OIL1.OUT;
OIL_1_DIO.0 := OIL1.OUT;
(* Network 13 *)
OIL2(EN := TRUE, MILL_ALR_STOP := MILL_ALR_STOP_2, MILL_ALR_STOP_VIRT := MILL_2.0, MILL_AUTO := MILL_AUTO_2, MILL_AUTO_VIRT := MILL_2.4, MILL_MAN := MILL_MAN_2, OIL_START := OIL_ST_START_2, SEPR_RUN := SEPR_RUN_2, OIL_STOP := OIL_ST_STOP_2, MILL_KM := MILL_RUN_2, OIL_KM_ERROR := OIL_2_DIO.1, SEPR_START_VIRT := MILL_2.1);
OIL_ST_RUN_2 := OIL2.OUT;
OIL_2_DIO.0 := OIL2.OUT;
(* Network 14 *)
MILL1(EN := TRUE, MILL_ALR_STOP := MILL_ALR_STOP_1, MILL_ALR_STOP_VIRT := MILL_1.0, MILL_AUTO := MILL_AUTO_1, MILL_AUTO_VIRT := MILL_1.4, MILL_MAN := SEPR_RUN_1, MILL_START := MILL_START_1, OIL_KM := OIL_ST_KM_1, MILL_ENC := MILL_ENC_1, MILL_STOP := MILL_STOP_1, FAN_KM := FAN_KM_1, MILL_KM_ERROR := MILL_1_DIO.1, SIMULATION := MILL_1_DIO.12, SEPR_START_VIRT := MILL_1.1, vaqtInduc := vaqtInduc, MILL_startTIME := MILL_1_startTIME, MILL_stopTIME := MILL_1_stopTIME, SEP_KM := SEPR_KM_1);
MILL_1_DIO.2 := MILL1.ALARM;
MILL_RUN_1 := MILL1.OUT;
MILL_1_DIO.0 := MILL1.OUT;
(* Network 15 *)
MILL2(EN := TRUE, MILL_ALR_STOP := MILL_ALR_STOP_2, MILL_ALR_STOP_VIRT := MILL_2.0, MILL_AUTO := MILL_AUTO_2, MILL_AUTO_VIRT := MILL_2.4, MILL_MAN := MILL_MAN_2, MILL_START := MILL_START_2, OIL_KM := OIL_ST_RUN_2, MILL_ENC := MILL_ENC_2, MILL_STOP := MILL_STOP_2, FAN_KM := FAN_RUN_2, MILL_KM_ERROR := MILL_2_DIO.1, SIMULATION := MILL_2_DIO.12, SEPR_START_VIRT := MILL_2.1, vaqtInduc := vaqtInduc, MILL_startTIME := MILL_2_startTIME, MILL_stopTIME := MILL_2_stopTIME, SEP_KM := SEPR_KM_2);
MILL_2_DIO.2 := MILL2.ALARM;
MILL_RUN_2 := MILL2.OUT;
MILL_2_DIO.0 := MILL2.OUT;
(* Network 16 *)
FAN1(EN := TRUE, MILL_ALR_STOP := MILL_ALR_STOP_1, MILL_ALR_STOP_VIRT := MILL_1.0, MILL_AUTO := MILL_AUTO_1, MILL_AUTO_VIRT := MILL_1.4, MILL_MAN := MILL_MAN_1, FAN_START := FAN_START_1, VIBRATOR_T := VIBRATOR1_T, FAN_STOP := FAN_STOP_1, MILL_KM := MILL_RUN_1, FAN_KM_ERROR := FAN_1_DIO.1, SEPR_START_VIRT := MILL_1.1, FAN_startTIME := FAN_1_startTIME, FAN_stopTIME := FAN_1_stopTIME);
FAN_1_DIO.2 := FAN1.ALARM;
FAN_RUN_1 := FAN1.OUT;
FAN_1_DIO.0 := FAN1.OUT;
(* Network 17 *)
FAN2(EN := TRUE, MILL_ALR_STOP := MILL_ALR_STOP_2, MILL_ALR_STOP_VIRT := MILL_2.0, MILL_AUTO := MILL_AUTO_2, MILL_AUTO_VIRT := MILL_2.4, MILL_MAN := MILL_MAN_2, FAN_START := FAN_START_2, VIBRATOR_T := VIBRATOR2_T, FAN_STOP := FAN_STOP_2, MILL_KM := MILL_RUN_2, FAN_KM_ERROR := FAN_2_DIO.1, SEPR_START_VIRT := MILL_2.1, FAN_startTIME := FAN_2_startTIME, FAN_stopTIME := FAN_2_stopTIME);
FAN_2_DIO.2 := FAN2.ALARM;
FAN_RUN_2 := FAN2.OUT;
FAN_2_DIO.0 := FAN2.OUT;
(* Network 18 *)
CONV1(EN := TRUE, MILL_ALR_STOP := MILL_ALR_STOP_1, MILL_ALR_STOP_VIRT := MILL_1.0, MILL_AUTO := MILL_AUTO_1, MILL_AUTO_VIRT := MILL_1.4, MILL_MAN := MILL_MAN_1, CONV_START := CONV_START_1, FAN_KM := FAN_RUN_1, MILL_KM := MILL_RUN_1, CONV_ENC := CONV_ENC_1, CONV_STOP := CONV_STOP_1, VIBRATOR_T := VIBRATOR1_T, CONV_KM_ERROR := CONV_1_DIO.1, SIMULATION := CONV_RUN_1, MATER_FULL := MATER_FULL_1, SEPR_START_VIRT := MILL_1.1, vaqtInduc := vaqtInduc);
CONV_1_DIO.2 := CONV1.ALARM;
CONV_RUN_1 := CONV1.OUT;
CONV_1_DIO.0 := CONV1.OUT;
(* Network 19 *)
CONV2(EN := TRUE, MILL_ALR_STOP := MILL_ALR_STOP_2, MILL_ALR_STOP_VIRT := MILL_2.0, MILL_AUTO := MILL_AUTO_2, MILL_AUTO_VIRT := MILL_2.4, MILL_MAN := MILL_MAN_2, CONV_START := CONV_START_2, FAN_KM := FAN_RUN_2, MILL_KM := MILL_RUN_2, CONV_ENC := CONV_ENC_2, CONV_STOP := CONV_STOP_2, VIBRATOR_T := VIBRATOR2_T, CONV_KM_ERROR := CONV_1_DIO.1, SIMULATION := CONV_RUN_2, MATER_FULL := MATER_FULL_1, SEPR_START_VIRT := MILL_2.1, vaqtInduc := vaqtInduc);
CONV_2_DIO.2 := CONV2.ALARM;
CONV_RUN_2 := CONV2.OUT;
CONV_2_DIO.0 := CONV2.OUT;
(* Network 20 *)
VIBRATOR1_T := NOT MILL_1.0 AND NOT MILL_ALR_STOP_1 AND (MILL_AUTO_1 OR MILL_MAN_1 OR MILL_1.4) AND (VIBR_START_1 OR VIBRATOR1_T OR CONV_RUN_1) AND VIBR_STOP_1 AND NOT TANK_MAX AND NOT MILL_1.3 AND OIL_ST_RUN_1 AND MILL_RUN_1;
(* Network 21 *)
VIBRATOR2_T := NOT MILL_2.0 AND NOT MILL_ALR_STOP_2 AND (MILL_AUTO_2 OR MILL_MAN_2 OR MILL_2.4) AND (VIBR_START_2 OR VIBRATOR2_T OR CONV_RUN_2) AND VIBR_STOP_2 AND NOT TANK_MAX AND NOT MILL_2.3 AND OIL_ST_RUN_2 AND MILL_RUN_2;
(* Network 22 *)
VALV_RUN_1 := NOT MILL_ALR_STOP_1 AND (MILL_AUTO_1 OR MILL_MAN_1 OR MILL_1.4) AND SEPR_KM_1 AND SEPR_RUN_1;
VALV_1_DIO.0 := VALV_RUN_1;
(* Network 23 *)
VALV_RUN_2 := NOT MILL_ALR_STOP_2 AND (MILL_AUTO_2 OR MILL_MAN_2 OR MILL_2.4) AND SEPR_KM_2 AND SEPR_RUN_2;
VALV_2_DIO.0 := VALV_RUN_2;
(* Network 24 *)
TON1(IN := NOT TON2.Q, PT := VAQT);
VIBR_RUN_1 := TON1.Q AND VIBRATOR1_T AND CONV_KM_1 AND NOT VIBR_1_DIO.1;
VIBR_1_DIO.0 := VIBR_RUN_1;
(* Network 25 *)
TON1(IN := NOT TON2.Q, PT := VAQT);
VIBR_RUN_2 := TON1.Q AND VIBRATOR2_T AND CONV_KM_2 AND NOT VIBR_2_DIO.1;
VIBR_2_DIO.0 := VIBR_RUN_2;
(* Network 26 *)
TON2(IN := TON1.Q, PT := VAQT);
(* Network 27 *)
(* Network 28 *)
_p1 := RESET_1 OR RESET_2 OR MILL_1.2 OR MILL_2.2 OR MILL_1.0;
IF _p1 THEN MILL_1.3 := FALSE; MILL_1.1 := FALSE; END_IF;
(* Network 29 *)
IF MILL_1.1 THEN MILL_1.3 := FALSE; END_IF;
(* Network 30 *)
IF MILL_1.3 THEN MILL_1.1 := FALSE; END_IF;
(* Network 31 *)
_p2 := RESET_1 OR RESET_2 OR MILL_1.2 OR MILL_2.2 OR MILL_2.0;
IF _p2 THEN MILL_2.3 := FALSE; MILL_2.1 := FALSE; END_IF;
(* Network 32 *)
IF MILL_2.1 THEN MILL_2.3 := FALSE; END_IF;
(* Network 33 *)
IF MILL_2.3 THEN MILL_2.1 := FALSE; END_IF;
(* Network 34 *)
END_PROGRAM

(* POU ELEV, LD *)
FUNCTION_BLOCK ELEV
VAR_INPUT
	EN : BOOL;
	MILL_ALR_STOP1: BOOL;
	MILL_ALR_STOP2: BOOL;
	MILL_ALR_STOP_VIRT1 : BOOL;
	MILL_ALR_STOP_VIRT2 : BOOL;
	MILL_AUTO1 : BOOL;
	MILL_AUTO2 : BOOL;
	MILL_AUTO_VIRT1 : BOOL;
	MILL_AUTO_VIRT2 : BOOL;
	TANK_MAX : BOOL;
	MILL_MAN1 : BOOL;
	MILL_MAN2 : BOOL;
	ELEV_START1 : BOOL;
	ELEV_START2 : BOOL;
	VIBR_RUN_1 : BOOL;
	VIBR_RUN_2 : BOOL;
	ELEV_ENC : BOOL;
	ELEV_STOP1 : BOOL;
	ELEV_STOP2 : BOOL;
	SHNK_KM1 : BOOL;
	SHNK_KM2 : BOOL;
	ELEV_KM_ERROR : BOOL;
	SIMULATION : BOOL := TRUE;
	SEPR_START_VIRT1 : BOOL;
	SEPR_START_VIRT2 : BOOL;
	vaqtInduc : WORD := 15;
	ELEV_startTIME : WORD;
	ELEV_stopTIME : WORD;
END_VAR

VAR_OUTPUT
	OUT : BOOL;
	ALARM : BOOL;
END_VAR
VAR
	INDUK1: INDUKTIV;
	INDUK2: INDUKTIV;
	OUT_MAN: BOOL;
	OUT_AUTO: BOOL;
	START_TON : TON;
	STOP_TOF : TOF;
	startTIME : TIME;
	stopTIME : TIME;
	L1: BOOL;
	L2: BOOL;
	ES: BOOL;
	EMERGENCY_STOP: BOOL;
	ALARM1 : BOOL;
	ALARM2 : BOOL;

	STOP: BOOL;
	ALLOW: BOOL;
	START_timer: BOOL;
	STOP_timer: BOOL;
	TTT : TP;
	L3: BOOL;
END_VAR
VAR (* helpers for the ST form of the networks *)
	_p1 : BOOL;
END_VAR
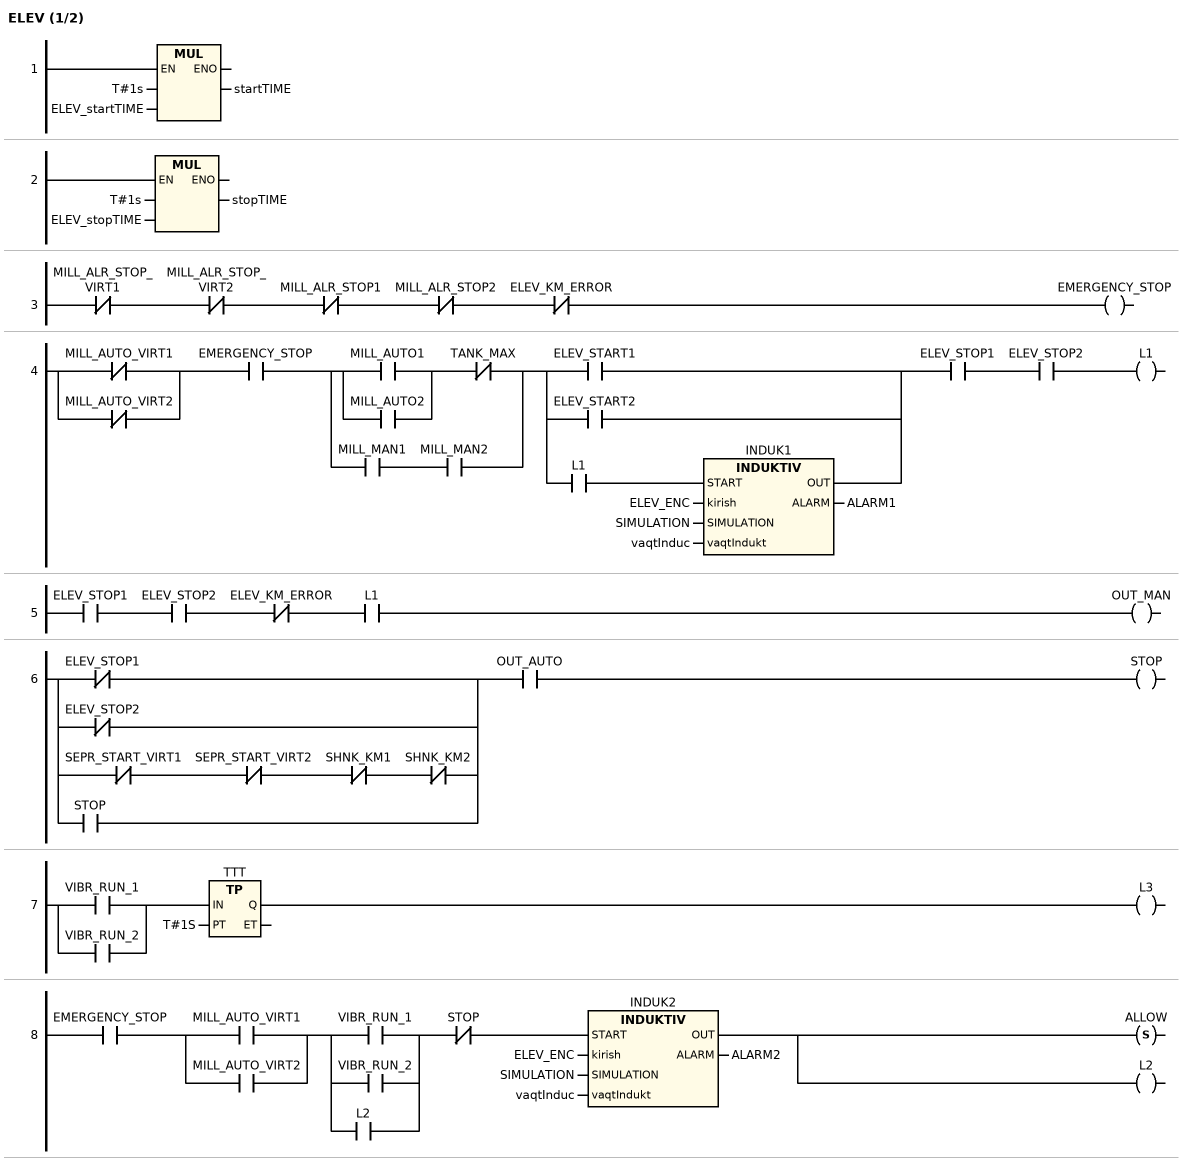
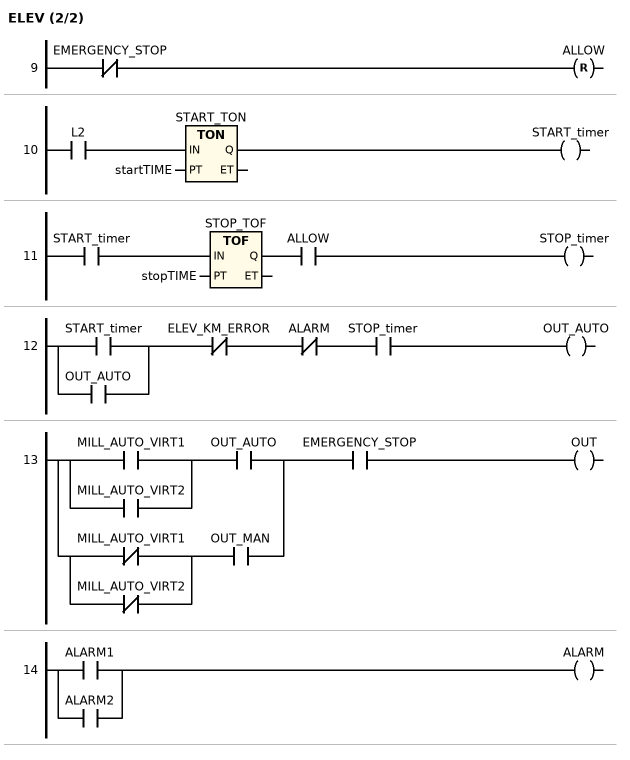
_LD_ (* Ladder Diagram *)
NETWORK 1
	*
		EN --- MUL(T#1s, ELEV_startTIME) => startTIME
NETWORK 2
	*
		EN --- MUL(T#1s, ELEV_stopTIME) => stopTIME
NETWORK 3
	[/MILL_ALR_STOP_VIRT1] - [/MILL_ALR_STOP_VIRT2] - [/MILL_ALR_STOP1] - [/MILL_ALR_STOP2] - [/ELEV_KM_ERROR] --- (EMERGENCY_STOP)
NETWORK 4
	{ [/MILL_AUTO_VIRT1] | [/MILL_AUTO_VIRT2] } - [EMERGENCY_STOP] - { { [MILL_AUTO1] | [MILL_AUTO2] } - [/TANK_MAX] | [MILL_MAN1] - [MILL_MAN2] } - { [ELEV_START1] | [ELEV_START2] | [L1] - INDUK1:INDUKTIV(START: *, kirish: ELEV_ENC, SIMULATION: SIMULATION, vaqtIndukt: vaqtInduc, ALARM => ALARM1) } - [ELEV_STOP1] - [ELEV_STOP2] --- (L1)
NETWORK 5
	[ELEV_STOP1] - [ELEV_STOP2] - [/ELEV_KM_ERROR] - [L1] --- (OUT_MAN)
NETWORK 6
	{ [/ELEV_STOP1] | [/ELEV_STOP2] | [/SEPR_START_VIRT1] - [/SEPR_START_VIRT2] - [/SHNK_KM1] - [/SHNK_KM2] | [STOP] } - [OUT_AUTO] --- (STOP)
NETWORK 7
	{ [VIBR_RUN_1] | [VIBR_RUN_2] } - TTT:TP(IN: *, PT: T#1S) --- (L3)
NETWORK 8
	[EMERGENCY_STOP] - { [MILL_AUTO_VIRT1] | [MILL_AUTO_VIRT2] } - { [VIBR_RUN_1] | [VIBR_RUN_2] | [L2] } - [/STOP] - INDUK2:INDUKTIV(START: *, kirish: ELEV_ENC, SIMULATION: SIMULATION, vaqtIndukt: vaqtInduc, ALARM => ALARM2) --- (S ALLOW) (L2)
NETWORK 9
	[/EMERGENCY_STOP] --- (R ALLOW)
NETWORK 10
	[L2] - START_TON:TON(IN: *, PT: startTIME) --- (START_timer)
NETWORK 11
	[START_timer] - STOP_TOF:TOF(IN: *, PT: stopTIME) - [ALLOW] --- (STOP_timer)
NETWORK 12
	{ [START_timer] | [OUT_AUTO] } - [/ELEV_KM_ERROR] - [/ALARM] - [STOP_timer] --- (OUT_AUTO)
NETWORK 13
	{ { [MILL_AUTO_VIRT1] | [MILL_AUTO_VIRT2] } - [OUT_AUTO] | { [/MILL_AUTO_VIRT1] | [/MILL_AUTO_VIRT2] } - [OUT_MAN] } - [EMERGENCY_STOP] --- (OUT)
NETWORK 14
	{ [ALARM1] | [ALARM2] } --- (ALARM)
_END_LD_
(* the same logic as Structured Text *)
(* Network 1 *)
startTIME := T#1s * ELEV_startTIME;
(* Network 2 *)
stopTIME := T#1s * ELEV_stopTIME;
(* Network 3 *)
EMERGENCY_STOP := NOT MILL_ALR_STOP_VIRT1 AND NOT MILL_ALR_STOP_VIRT2 AND NOT MILL_ALR_STOP1 AND NOT MILL_ALR_STOP2 AND NOT ELEV_KM_ERROR;
(* Network 4 *)
_p1 := (NOT MILL_AUTO_VIRT1 OR NOT MILL_AUTO_VIRT2) AND EMERGENCY_STOP AND ((MILL_AUTO1 OR MILL_AUTO2) AND NOT TANK_MAX OR MILL_MAN1 AND MILL_MAN2);
INDUK1(START := _p1 AND L1, kirish := ELEV_ENC, SIMULATION := SIMULATION, vaqtIndukt := vaqtInduc);
ALARM1 := INDUK1.ALARM;
L1 := (_p1 AND ELEV_START1 OR _p1 AND ELEV_START2 OR INDUK1.OUT) AND ELEV_STOP1 AND ELEV_STOP2;
(* Network 5 *)
OUT_MAN := ELEV_STOP1 AND ELEV_STOP2 AND NOT ELEV_KM_ERROR AND L1;
(* Network 6 *)
STOP := (NOT ELEV_STOP1 OR NOT ELEV_STOP2 OR NOT SEPR_START_VIRT1 AND NOT SEPR_START_VIRT2 AND NOT SHNK_KM1 AND NOT SHNK_KM2 OR STOP) AND OUT_AUTO;
(* Network 7 *)
TTT(IN := VIBR_RUN_1 OR VIBR_RUN_2, PT := T#1S);
L3 := TTT.Q;
(* Network 8 *)
INDUK2(START := EMERGENCY_STOP AND (MILL_AUTO_VIRT1 OR MILL_AUTO_VIRT2) AND (VIBR_RUN_1 OR VIBR_RUN_2 OR L2) AND NOT STOP, kirish := ELEV_ENC, SIMULATION := SIMULATION, vaqtIndukt := vaqtInduc);
ALARM2 := INDUK2.ALARM;
IF INDUK2.OUT THEN ALLOW := TRUE; END_IF;
L2 := INDUK2.OUT;
(* Network 9 *)
IF NOT EMERGENCY_STOP THEN ALLOW := FALSE; END_IF;
(* Network 10 *)
START_TON(IN := L2, PT := startTIME);
START_timer := START_TON.Q;
(* Network 11 *)
STOP_TOF(IN := START_timer, PT := stopTIME);
STOP_timer := STOP_TOF.Q AND ALLOW;
(* Network 12 *)
OUT_AUTO := (START_timer OR OUT_AUTO) AND NOT ELEV_KM_ERROR AND NOT ALARM AND STOP_timer;
(* Network 13 *)
OUT := ((MILL_AUTO_VIRT1 OR MILL_AUTO_VIRT2) AND OUT_AUTO OR (NOT MILL_AUTO_VIRT1 OR NOT MILL_AUTO_VIRT2) AND OUT_MAN) AND EMERGENCY_STOP;
(* Network 14 *)
ALARM := ALARM1 OR ALARM2;
END_FUNCTION_BLOCK

(* POU INDUKTIV, CFC *)
FUNCTION_BLOCK INDUKTIV
VAR_IN_OUT

	(*RESET : BOOL;*)

END_VAR
VAR_INPUT
	START : BOOL;
	kirish : BOOL;
	SIMULATION : BOOL;
	vaqtIndukt : WORD := 15;
END_VAR

VAR_OUTPUT

	OUT : BOOL;
	ALARM : BOOL;
END_VAR
VAR
	ton1: TON;
	vaqt : TIME;
	ton2: TON;
	TP1: TP;
	TP2: TP;


END_VAR
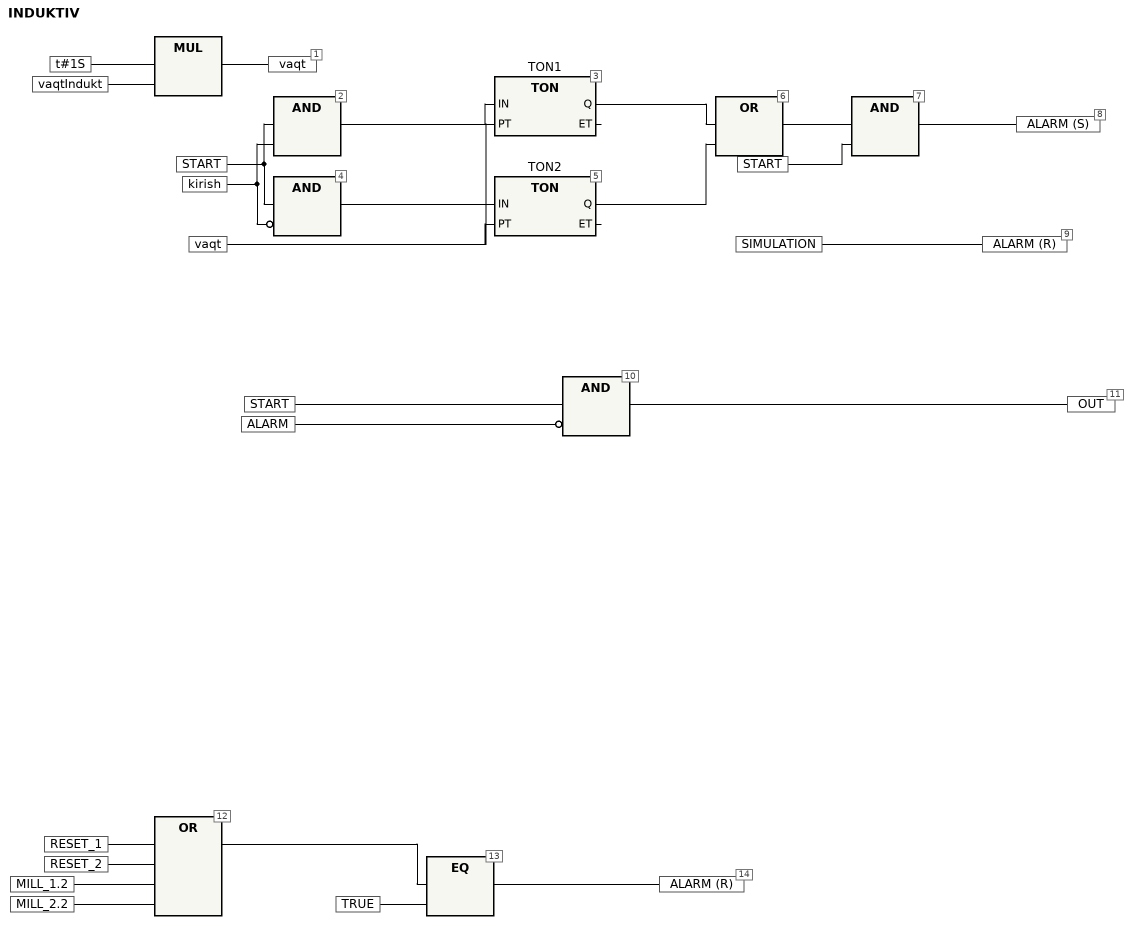
_CFC_ (* Continuous Function Chart, elements in execution order *)
#0 MUL(t#1S, vaqtIndukt)
#1 vaqt <= #0
#2 AND(START, kirish)
#3 TON1:TON(IN: #2, PT: vaqt)
#4 AND(START, NOT kirish)
#5 TON2:TON(IN: #4, PT: vaqt)
#6 OR(#3.Q, #5.Q)
#7 AND(#6, START)
#8 S ALARM <= #7
#9 R ALARM <= SIMULATION
#10 AND(START, NOT ALARM)
#11 OUT <= #10
#12 OR(RESET_1, RESET_2, MILL_1.2, MILL_2.2)
#13 EQ(#12, TRUE)
#14 R ALARM <= #13
_END_CFC_
(* the same logic as Structured Text *)
vaqt := t#1S * vaqtIndukt;
TON1(IN := START AND kirish, PT := vaqt);
TON2(IN := START AND NOT kirish, PT := vaqt);
IF (TON1.Q OR TON2.Q) AND START THEN ALARM := TRUE; END_IF;
IF SIMULATION THEN ALARM := FALSE; END_IF;
OUT := START AND NOT ALARM;
IF (RESET_1 OR RESET_2 OR MILL_1.2 OR MILL_2.2) = TRUE THEN ALARM := FALSE; END_IF;
END_FUNCTION_BLOCK

(* POU SHNEK, LD *)
FUNCTION_BLOCK SHNEK
VAR_INPUT
	EN : BOOL;
	MILL_ALR_STOP: BOOL;
	MILL_ALR_STOP_VIRT : BOOL;
	MILL_AUTO : BOOL;
	MILL_AUTO_VIRT : BOOL;
	MILL_MAN : BOOL;
	SHNK_START : BOOL;
	SEP_RUN : BOOL;
	ELEV_KM : BOOL;
	SHNK_ENC : BOOL;
	SHNK_STOP : BOOL;
	SHNK_SIKL_KM : BOOL;
	SHNK_KM_ERROR : BOOL;
	SIMULATION : BOOL := TRUE;
	SEPR_START_VIRT : BOOL;
	vaqtInduc : WORD := 15;
	SHNK_startTIME : WORD;
	SHNK_stopTIME : WORD;
END_VAR

VAR_OUTPUT
	OUT : BOOL;
	ALARM : BOOL;
END_VAR
VAR
	INDUK1: INDUKTIV;
	INDUK2: INDUKTIV;
	OUT_MAN: BOOL;
	OUT_AUTO: BOOL;
	START_TON : TON;
	STOP_TOF : TOF;
	startTIME : TIME;
	stopTIME : TIME;
	L1: BOOL;
	L2: BOOL;
	ES: BOOL;
	EMERGENCY_STOP: BOOL;
	ALARM1 : BOOL;
	ALARM2 : BOOL;

	STOP: BOOL;
	ALLOW: BOOL;
	START_timer: BOOL;
	STOP_timer: BOOL;
	TTT : TP;
END_VAR
VAR (* helpers for the ST form of the networks *)
	_p1 : BOOL;
END_VAR
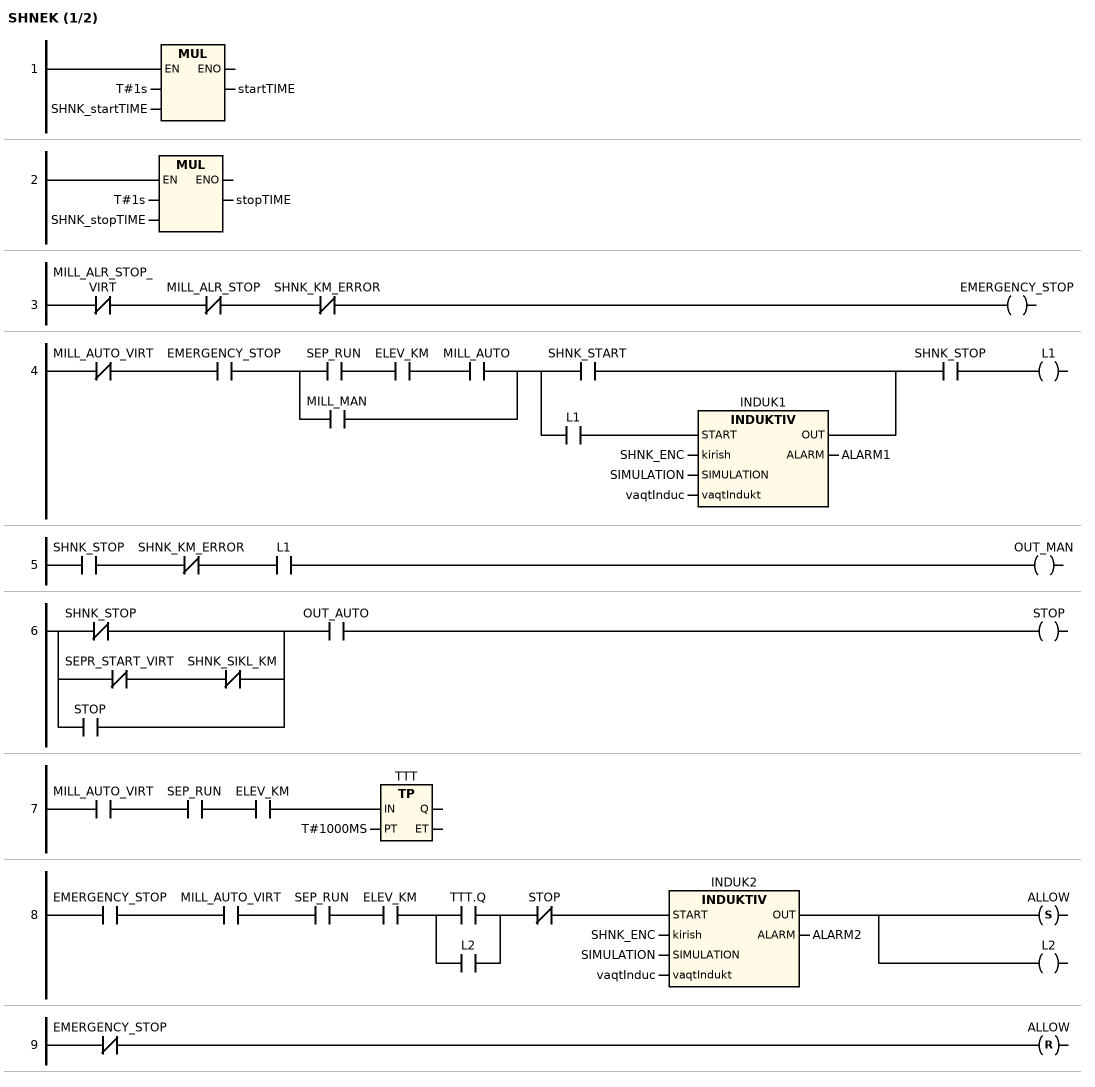
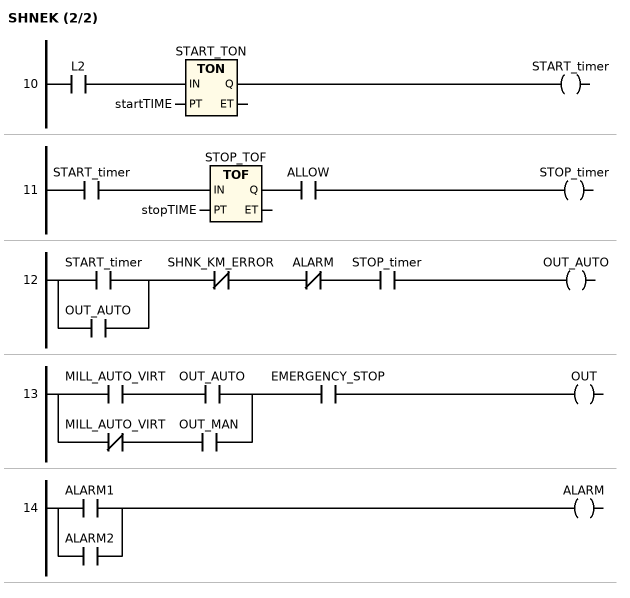
_LD_ (* Ladder Diagram *)
NETWORK 1
	*
		EN --- MUL(T#1s, SHNK_startTIME) => startTIME
NETWORK 2
	*
		EN --- MUL(T#1s, SHNK_stopTIME) => stopTIME
NETWORK 3
	[/MILL_ALR_STOP_VIRT] - [/MILL_ALR_STOP] - [/SHNK_KM_ERROR] --- (EMERGENCY_STOP)
NETWORK 4
	[/MILL_AUTO_VIRT] - [EMERGENCY_STOP] - { [SEP_RUN] - [ELEV_KM] - [MILL_AUTO] | [MILL_MAN] } - { [SHNK_START] | [L1] - INDUK1:INDUKTIV(START: *, kirish: SHNK_ENC, SIMULATION: SIMULATION, vaqtIndukt: vaqtInduc, ALARM => ALARM1) } - [SHNK_STOP] --- (L1)
NETWORK 5
	[SHNK_STOP] - [/SHNK_KM_ERROR] - [L1] --- (OUT_MAN)
NETWORK 6
	{ [/SHNK_STOP] | [/SEPR_START_VIRT] - [/SHNK_SIKL_KM] | [STOP] } - [OUT_AUTO] --- (STOP)
NETWORK 7
	[MILL_AUTO_VIRT] - [SEP_RUN] - [ELEV_KM] - TTT:TP(IN: *, PT: T#1000MS)
NETWORK 8
	[EMERGENCY_STOP] - [MILL_AUTO_VIRT] - [SEP_RUN] - [ELEV_KM] - { [TTT.Q] | [L2] } - [/STOP] - INDUK2:INDUKTIV(START: *, kirish: SHNK_ENC, SIMULATION: SIMULATION, vaqtIndukt: vaqtInduc, ALARM => ALARM2) --- (S ALLOW) (L2)
NETWORK 9
	[/EMERGENCY_STOP] --- (R ALLOW)
NETWORK 10
	[L2] - START_TON:TON(IN: *, PT: startTIME) --- (START_timer)
NETWORK 11
	[START_timer] - STOP_TOF:TOF(IN: *, PT: stopTIME) - [ALLOW] --- (STOP_timer)
NETWORK 12
	{ [START_timer] | [OUT_AUTO] } - [/SHNK_KM_ERROR] - [/ALARM] - [STOP_timer] --- (OUT_AUTO)
NETWORK 13
	{ [MILL_AUTO_VIRT] - [OUT_AUTO] | [/MILL_AUTO_VIRT] - [OUT_MAN] } - [EMERGENCY_STOP] --- (OUT)
NETWORK 14
	{ [ALARM1] | [ALARM2] } --- (ALARM)
_END_LD_
(* the same logic as Structured Text *)
(* Network 1 *)
startTIME := T#1s * SHNK_startTIME;
(* Network 2 *)
stopTIME := T#1s * SHNK_stopTIME;
(* Network 3 *)
EMERGENCY_STOP := NOT MILL_ALR_STOP_VIRT AND NOT MILL_ALR_STOP AND NOT SHNK_KM_ERROR;
(* Network 4 *)
_p1 := NOT MILL_AUTO_VIRT AND EMERGENCY_STOP AND (SEP_RUN AND ELEV_KM AND MILL_AUTO OR MILL_MAN);
INDUK1(START := _p1 AND L1, kirish := SHNK_ENC, SIMULATION := SIMULATION, vaqtIndukt := vaqtInduc);
ALARM1 := INDUK1.ALARM;
L1 := (_p1 AND SHNK_START OR INDUK1.OUT) AND SHNK_STOP;
(* Network 5 *)
OUT_MAN := SHNK_STOP AND NOT SHNK_KM_ERROR AND L1;
(* Network 6 *)
STOP := (NOT SHNK_STOP OR NOT SEPR_START_VIRT AND NOT SHNK_SIKL_KM OR STOP) AND OUT_AUTO;
(* Network 7 *)
TTT(IN := MILL_AUTO_VIRT AND SEP_RUN AND ELEV_KM, PT := T#1000MS);
(* Network 8 *)
INDUK2(START := EMERGENCY_STOP AND MILL_AUTO_VIRT AND SEP_RUN AND ELEV_KM AND (TTT.Q OR L2) AND NOT STOP, kirish := SHNK_ENC, SIMULATION := SIMULATION, vaqtIndukt := vaqtInduc);
ALARM2 := INDUK2.ALARM;
IF INDUK2.OUT THEN ALLOW := TRUE; END_IF;
L2 := INDUK2.OUT;
(* Network 9 *)
IF NOT EMERGENCY_STOP THEN ALLOW := FALSE; END_IF;
(* Network 10 *)
START_TON(IN := L2, PT := startTIME);
START_timer := START_TON.Q;
(* Network 11 *)
STOP_TOF(IN := START_timer, PT := stopTIME);
STOP_timer := STOP_TOF.Q AND ALLOW;
(* Network 12 *)
OUT_AUTO := (START_timer OR OUT_AUTO) AND NOT SHNK_KM_ERROR AND NOT ALARM AND STOP_timer;
(* Network 13 *)
OUT := (MILL_AUTO_VIRT AND OUT_AUTO OR NOT MILL_AUTO_VIRT AND OUT_MAN) AND EMERGENCY_STOP;
(* Network 14 *)
ALARM := ALARM1 OR ALARM2;
END_FUNCTION_BLOCK

(* POU SHNEK_SIKL, LD *)
FUNCTION_BLOCK SHNEK_SIKL
VAR_INPUT
	EN : BOOL;
	MILL_ALR_STOP: BOOL;
	MILL_ALR_STOP_VIRT : BOOL;
	MILL_AUTO : BOOL;
	MILL_AUTO_VIRT : BOOL;
	MILL_MAN : BOOL;
	SHNK_SIKL_START : BOOL;
	SHNK_KM : BOOL;
	SHNK_SIKL_ENC : BOOL;
	SHNK_SIKL_STOP : BOOL;
	STAR_1_KM : BOOL;
	SHNK_SIKL_KM_ERROR : BOOL;
	SIMULATION : BOOL := TRUE;
	SEPR_START_VIRT : BOOL;
	vaqtInduc : WORD := 15;
	SHNK_SIKL_startTIME : WORD;
	SHNK_SIKL_stopTIME : WORD;
END_VAR

VAR_OUTPUT
	OUT : BOOL;
	ALARM : BOOL;
END_VAR
VAR
	INDUK1: INDUKTIV;
	INDUK2: INDUKTIV;
	OUT_MAN: BOOL;
	OUT_AUTO: BOOL;
	START_TON : TON;
	STOP_TOF : TOF;
	startTIME : TIME;
	stopTIME : TIME;
	L1: BOOL;
	L2: BOOL;
	ES: BOOL;
	EMERGENCY_STOP: BOOL;
	ALARM1 : BOOL;
	ALARM2 : BOOL;

	STOP: BOOL;
	ALLOW: BOOL;
	START_timer: BOOL;
	STOP_timer: BOOL;
	TTT : TP;
END_VAR
VAR (* helpers for the ST form of the networks *)
	_p1 : BOOL;
END_VAR
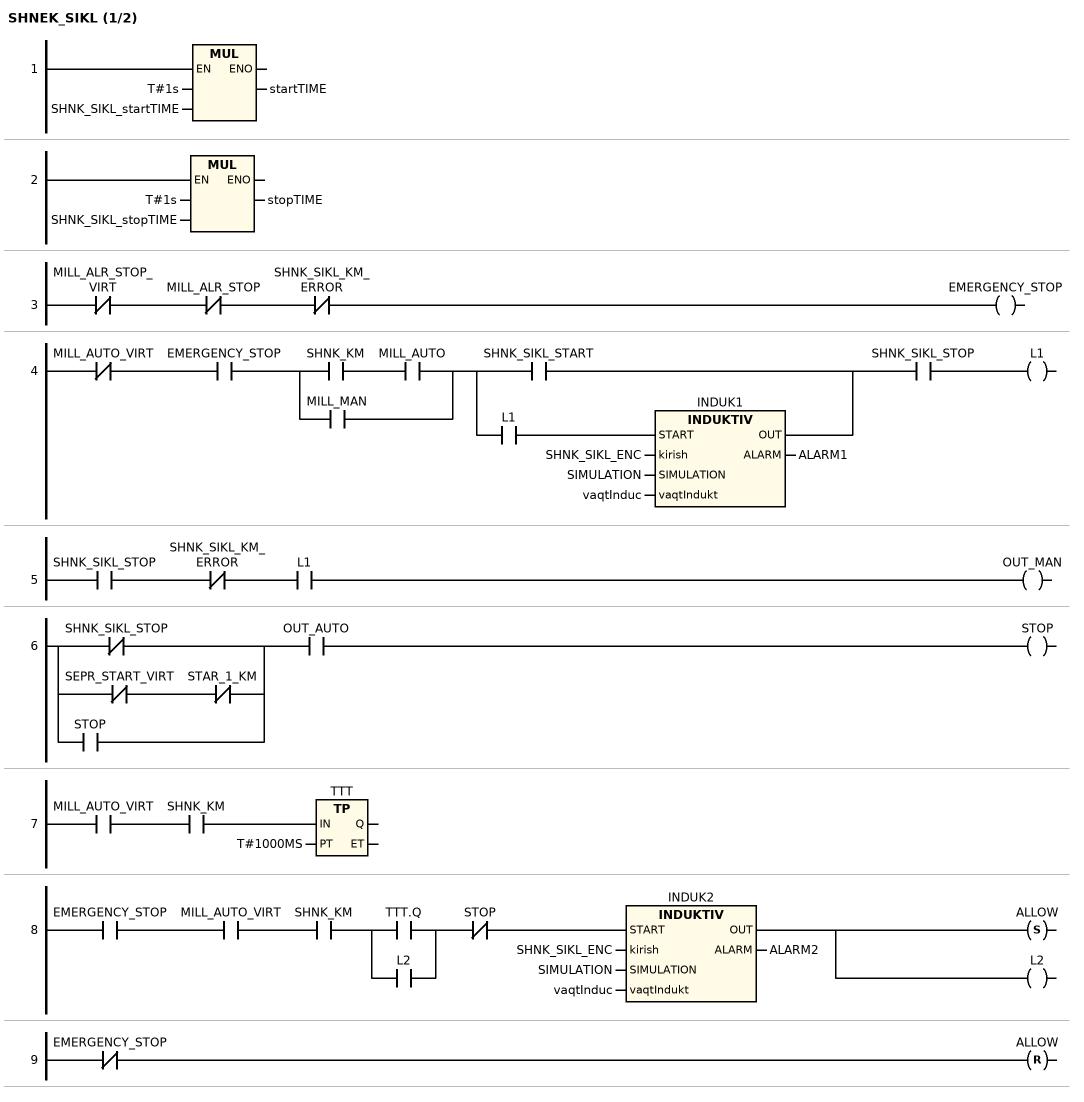
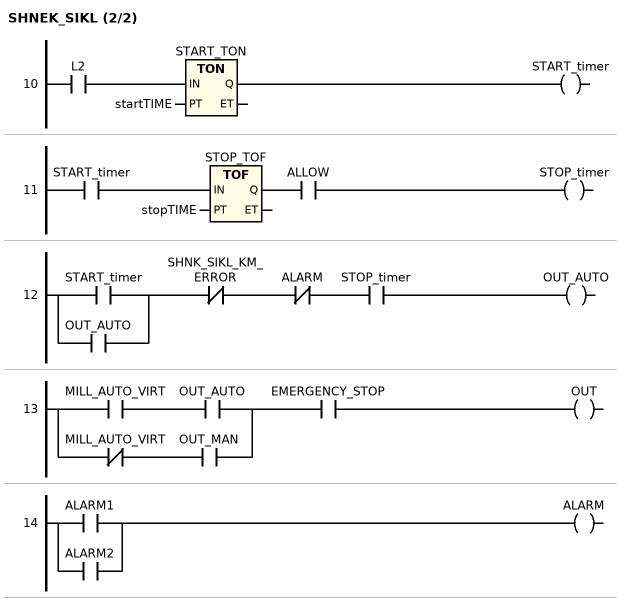
_LD_ (* Ladder Diagram *)
NETWORK 1
	*
		EN --- MUL(T#1s, SHNK_SIKL_startTIME) => startTIME
NETWORK 2
	*
		EN --- MUL(T#1s, SHNK_SIKL_stopTIME) => stopTIME
NETWORK 3
	[/MILL_ALR_STOP_VIRT] - [/MILL_ALR_STOP] - [/SHNK_SIKL_KM_ERROR] --- (EMERGENCY_STOP)
NETWORK 4
	[/MILL_AUTO_VIRT] - [EMERGENCY_STOP] - { [SHNK_KM] - [MILL_AUTO] | [MILL_MAN] } - { [SHNK_SIKL_START] | [L1] - INDUK1:INDUKTIV(START: *, kirish: SHNK_SIKL_ENC, SIMULATION: SIMULATION, vaqtIndukt: vaqtInduc, ALARM => ALARM1) } - [SHNK_SIKL_STOP] --- (L1)
NETWORK 5
	[SHNK_SIKL_STOP] - [/SHNK_SIKL_KM_ERROR] - [L1] --- (OUT_MAN)
NETWORK 6
	{ [/SHNK_SIKL_STOP] | [/SEPR_START_VIRT] - [/STAR_1_KM] | [STOP] } - [OUT_AUTO] --- (STOP)
NETWORK 7
	[MILL_AUTO_VIRT] - [SHNK_KM] - TTT:TP(IN: *, PT: T#1000MS)
NETWORK 8
	[EMERGENCY_STOP] - [MILL_AUTO_VIRT] - [SHNK_KM] - { [TTT.Q] | [L2] } - [/STOP] - INDUK2:INDUKTIV(START: *, kirish: SHNK_SIKL_ENC, SIMULATION: SIMULATION, vaqtIndukt: vaqtInduc, ALARM => ALARM2) --- (S ALLOW) (L2)
NETWORK 9
	[/EMERGENCY_STOP] --- (R ALLOW)
NETWORK 10
	[L2] - START_TON:TON(IN: *, PT: startTIME) --- (START_timer)
NETWORK 11
	[START_timer] - STOP_TOF:TOF(IN: *, PT: stopTIME) - [ALLOW] --- (STOP_timer)
NETWORK 12
	{ [START_timer] | [OUT_AUTO] } - [/SHNK_SIKL_KM_ERROR] - [/ALARM] - [STOP_timer] --- (OUT_AUTO)
NETWORK 13
	{ [MILL_AUTO_VIRT] - [OUT_AUTO] | [/MILL_AUTO_VIRT] - [OUT_MAN] } - [EMERGENCY_STOP] --- (OUT)
NETWORK 14
	{ [ALARM1] | [ALARM2] } --- (ALARM)
_END_LD_
(* the same logic as Structured Text *)
(* Network 1 *)
startTIME := T#1s * SHNK_SIKL_startTIME;
(* Network 2 *)
stopTIME := T#1s * SHNK_SIKL_stopTIME;
(* Network 3 *)
EMERGENCY_STOP := NOT MILL_ALR_STOP_VIRT AND NOT MILL_ALR_STOP AND NOT SHNK_SIKL_KM_ERROR;
(* Network 4 *)
_p1 := NOT MILL_AUTO_VIRT AND EMERGENCY_STOP AND (SHNK_KM AND MILL_AUTO OR MILL_MAN);
INDUK1(START := _p1 AND L1, kirish := SHNK_SIKL_ENC, SIMULATION := SIMULATION, vaqtIndukt := vaqtInduc);
ALARM1 := INDUK1.ALARM;
L1 := (_p1 AND SHNK_SIKL_START OR INDUK1.OUT) AND SHNK_SIKL_STOP;
(* Network 5 *)
OUT_MAN := SHNK_SIKL_STOP AND NOT SHNK_SIKL_KM_ERROR AND L1;
(* Network 6 *)
STOP := (NOT SHNK_SIKL_STOP OR NOT SEPR_START_VIRT AND NOT STAR_1_KM OR STOP) AND OUT_AUTO;
(* Network 7 *)
TTT(IN := MILL_AUTO_VIRT AND SHNK_KM, PT := T#1000MS);
(* Network 8 *)
INDUK2(START := EMERGENCY_STOP AND MILL_AUTO_VIRT AND SHNK_KM AND (TTT.Q OR L2) AND NOT STOP, kirish := SHNK_SIKL_ENC, SIMULATION := SIMULATION, vaqtIndukt := vaqtInduc);
ALARM2 := INDUK2.ALARM;
IF INDUK2.OUT THEN ALLOW := TRUE; END_IF;
L2 := INDUK2.OUT;
(* Network 9 *)
IF NOT EMERGENCY_STOP THEN ALLOW := FALSE; END_IF;
(* Network 10 *)
START_TON(IN := L2, PT := startTIME);
START_timer := START_TON.Q;
(* Network 11 *)
STOP_TOF(IN := START_timer, PT := stopTIME);
STOP_timer := STOP_TOF.Q AND ALLOW;
(* Network 12 *)
OUT_AUTO := (START_timer OR OUT_AUTO) AND NOT SHNK_SIKL_KM_ERROR AND NOT ALARM AND STOP_timer;
(* Network 13 *)
OUT := (MILL_AUTO_VIRT AND OUT_AUTO OR NOT MILL_AUTO_VIRT AND OUT_MAN) AND EMERGENCY_STOP;
(* Network 14 *)
ALARM := ALARM1 OR ALARM2;
END_FUNCTION_BLOCK

(* POU STAR_1, LD *)
FUNCTION_BLOCK STAR_1
VAR_INPUT
	EN : BOOL;
	MILL_ALR_STOP: BOOL;
	MILL_ALR_STOP_VIRT : BOOL;
	MILL_AUTO : BOOL;
	MILL_AUTO_VIRT : BOOL;
	MILL_MAN : BOOL;
	STAR_START : BOOL;
	SHNK_SIKL_KM : BOOL;
	STAR_ENC : BOOL;
	STAR_STOP : BOOL;
	STAR_2_KM : BOOL;
	STAR_KM_ERROR : BOOL;
	SIMULATION : BOOL := TRUE;
	SEPR_START_VIRT : BOOL;
	vaqtInduc : WORD := 15;
	STAR_startTIME : WORD;
	STAR_stopTIME : WORD;
END_VAR

VAR_OUTPUT
	OUT : BOOL;
	ALARM : BOOL;
END_VAR
VAR
	INDUK1: INDUKTIV;
	INDUK2: INDUKTIV;
	OUT_MAN: BOOL;
	OUT_AUTO: BOOL;
	START_TON : TON;
	STOP_TOF : TOF;
	startTIME : TIME;
	stopTIME : TIME;
	L1: BOOL;
	L2: BOOL;
	ES: BOOL;
	EMERGENCY_STOP: BOOL;
	ALARM1 : BOOL;
	ALARM2 : BOOL;

	STOP: BOOL;
	ALLOW: BOOL;
	START_timer: BOOL;
	STOP_timer: BOOL;
	TTT : TP;
END_VAR
VAR (* helpers for the ST form of the networks *)
	_p1 : BOOL;
END_VAR
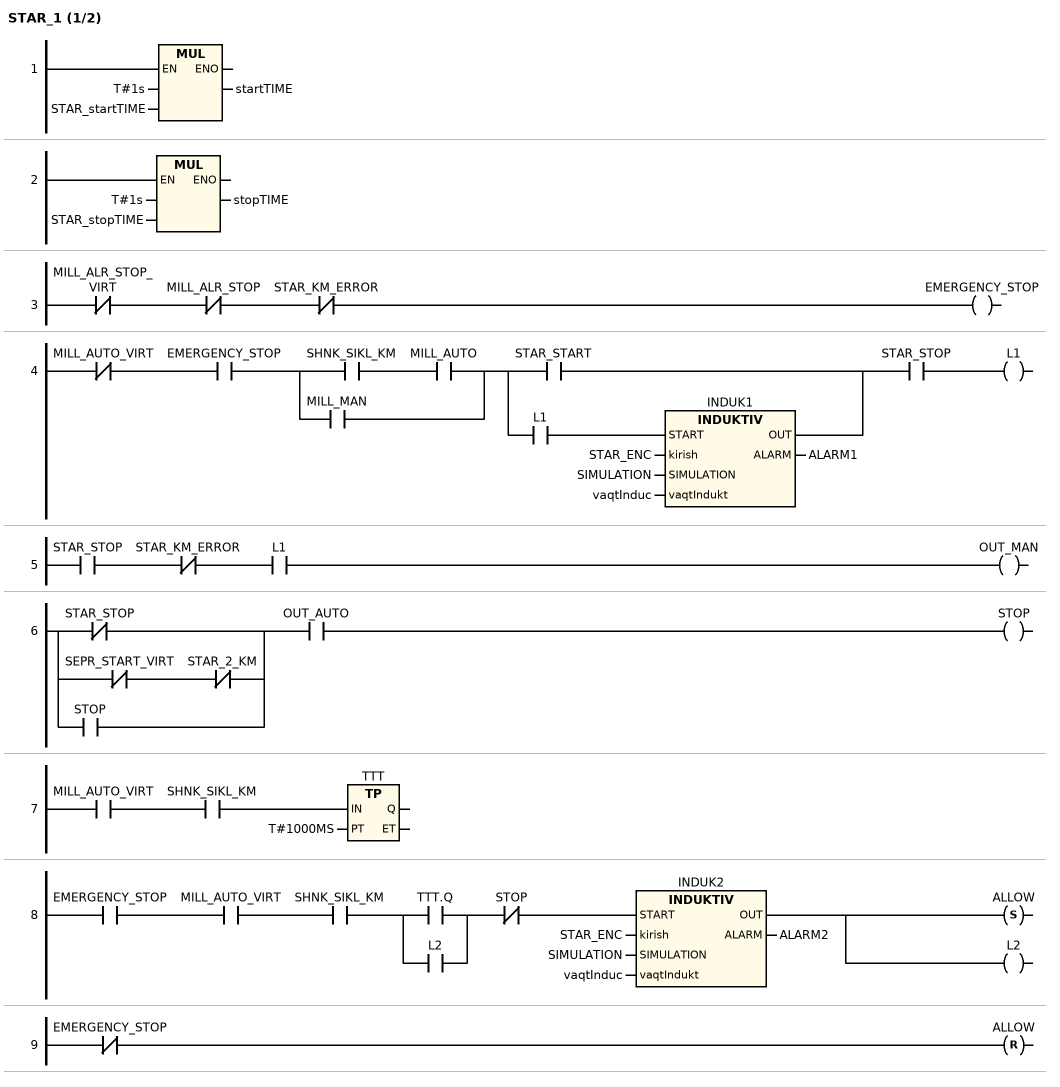
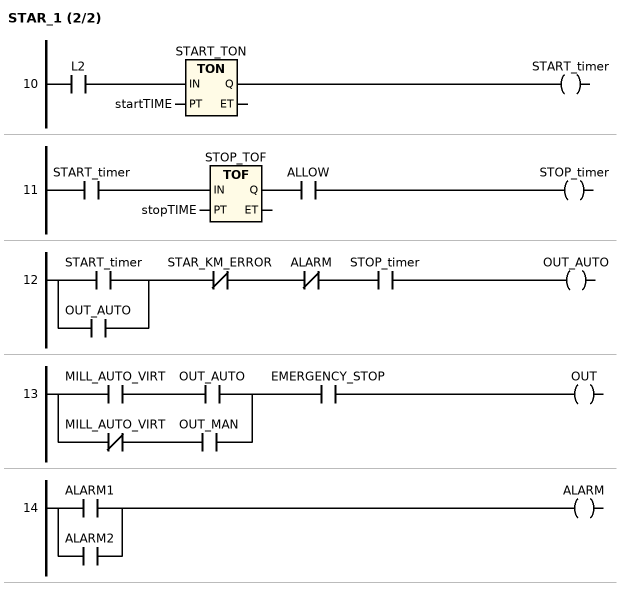
_LD_ (* Ladder Diagram *)
NETWORK 1
	*
		EN --- MUL(T#1s, STAR_startTIME) => startTIME
NETWORK 2
	*
		EN --- MUL(T#1s, STAR_stopTIME) => stopTIME
NETWORK 3
	[/MILL_ALR_STOP_VIRT] - [/MILL_ALR_STOP] - [/STAR_KM_ERROR] --- (EMERGENCY_STOP)
NETWORK 4
	[/MILL_AUTO_VIRT] - [EMERGENCY_STOP] - { [SHNK_SIKL_KM] - [MILL_AUTO] | [MILL_MAN] } - { [STAR_START] | [L1] - INDUK1:INDUKTIV(START: *, kirish: STAR_ENC, SIMULATION: SIMULATION, vaqtIndukt: vaqtInduc, ALARM => ALARM1) } - [STAR_STOP] --- (L1)
NETWORK 5
	[STAR_STOP] - [/STAR_KM_ERROR] - [L1] --- (OUT_MAN)
NETWORK 6
	{ [/STAR_STOP] | [/SEPR_START_VIRT] - [/STAR_2_KM] | [STOP] } - [OUT_AUTO] --- (STOP)
NETWORK 7
	[MILL_AUTO_VIRT] - [SHNK_SIKL_KM] - TTT:TP(IN: *, PT: T#1000MS)
NETWORK 8
	[EMERGENCY_STOP] - [MILL_AUTO_VIRT] - [SHNK_SIKL_KM] - { [TTT.Q] | [L2] } - [/STOP] - INDUK2:INDUKTIV(START: *, kirish: STAR_ENC, SIMULATION: SIMULATION, vaqtIndukt: vaqtInduc, ALARM => ALARM2) --- (S ALLOW) (L2)
NETWORK 9
	[/EMERGENCY_STOP] --- (R ALLOW)
NETWORK 10
	[L2] - START_TON:TON(IN: *, PT: startTIME) --- (START_timer)
NETWORK 11
	[START_timer] - STOP_TOF:TOF(IN: *, PT: stopTIME) - [ALLOW] --- (STOP_timer)
NETWORK 12
	{ [START_timer] | [OUT_AUTO] } - [/STAR_KM_ERROR] - [/ALARM] - [STOP_timer] --- (OUT_AUTO)
NETWORK 13
	{ [MILL_AUTO_VIRT] - [OUT_AUTO] | [/MILL_AUTO_VIRT] - [OUT_MAN] } - [EMERGENCY_STOP] --- (OUT)
NETWORK 14
	{ [ALARM1] | [ALARM2] } --- (ALARM)
_END_LD_
(* the same logic as Structured Text *)
(* Network 1 *)
startTIME := T#1s * STAR_startTIME;
(* Network 2 *)
stopTIME := T#1s * STAR_stopTIME;
(* Network 3 *)
EMERGENCY_STOP := NOT MILL_ALR_STOP_VIRT AND NOT MILL_ALR_STOP AND NOT STAR_KM_ERROR;
(* Network 4 *)
_p1 := NOT MILL_AUTO_VIRT AND EMERGENCY_STOP AND (SHNK_SIKL_KM AND MILL_AUTO OR MILL_MAN);
INDUK1(START := _p1 AND L1, kirish := STAR_ENC, SIMULATION := SIMULATION, vaqtIndukt := vaqtInduc);
ALARM1 := INDUK1.ALARM;
L1 := (_p1 AND STAR_START OR INDUK1.OUT) AND STAR_STOP;
(* Network 5 *)
OUT_MAN := STAR_STOP AND NOT STAR_KM_ERROR AND L1;
(* Network 6 *)
STOP := (NOT STAR_STOP OR NOT SEPR_START_VIRT AND NOT STAR_2_KM OR STOP) AND OUT_AUTO;
(* Network 7 *)
TTT(IN := MILL_AUTO_VIRT AND SHNK_SIKL_KM, PT := T#1000MS);
(* Network 8 *)
INDUK2(START := EMERGENCY_STOP AND MILL_AUTO_VIRT AND SHNK_SIKL_KM AND (TTT.Q OR L2) AND NOT STOP, kirish := STAR_ENC, SIMULATION := SIMULATION, vaqtIndukt := vaqtInduc);
ALARM2 := INDUK2.ALARM;
IF INDUK2.OUT THEN ALLOW := TRUE; END_IF;
L2 := INDUK2.OUT;
(* Network 9 *)
IF NOT EMERGENCY_STOP THEN ALLOW := FALSE; END_IF;
(* Network 10 *)
START_TON(IN := L2, PT := startTIME);
START_timer := START_TON.Q;
(* Network 11 *)
STOP_TOF(IN := START_timer, PT := stopTIME);
STOP_timer := STOP_TOF.Q AND ALLOW;
(* Network 12 *)
OUT_AUTO := (START_timer OR OUT_AUTO) AND NOT STAR_KM_ERROR AND NOT ALARM AND STOP_timer;
(* Network 13 *)
OUT := (MILL_AUTO_VIRT AND OUT_AUTO OR NOT MILL_AUTO_VIRT AND OUT_MAN) AND EMERGENCY_STOP;
(* Network 14 *)
ALARM := ALARM1 OR ALARM2;
END_FUNCTION_BLOCK

(* POU STAR_2, LD *)
FUNCTION_BLOCK STAR_2
VAR_INPUT
	EN : BOOL;
	MILL_ALR_STOP: BOOL;
	MILL_ALR_STOP_VIRT : BOOL;
	MILL_AUTO : BOOL;
	MILL_AUTO_VIRT : BOOL;
	MILL_MAN : BOOL;
	STAR_START : BOOL;
	STAR_1_KM : BOOL;
	STAR_ENC : BOOL;
	STAR_STOP : BOOL;
	OIL_KM : BOOL;
	STAR_KM_ERROR : BOOL;
	SIMULATION : BOOL := TRUE;
	vaqtInduc : WORD := 15;
	STAR_startTIME : WORD;
	STAR_stopTIME : WORD;
END_VAR

VAR_OUTPUT
	OUT : BOOL;
	ALARM : BOOL;
END_VAR
VAR
	INDUK1: INDUKTIV;
	INDUK2: INDUKTIV;
	OUT_MAN: BOOL;
	OUT_AUTO: BOOL;
	START_TON : TON;
	STOP_TOF : TOF;
	startTIME : TIME;
	stopTIME : TIME;
	L1: BOOL;
	L2: BOOL;
	ES: BOOL;
	EMERGENCY_STOP: BOOL;
	ALARM1 : BOOL;
	ALARM2 : BOOL;

	STOP: BOOL;
	ALLOW: BOOL;
	START_timer: BOOL;
	STOP_timer: BOOL;
	TTT : TP;
END_VAR
VAR (* helpers for the ST form of the networks *)
	_p1 : BOOL;
END_VAR
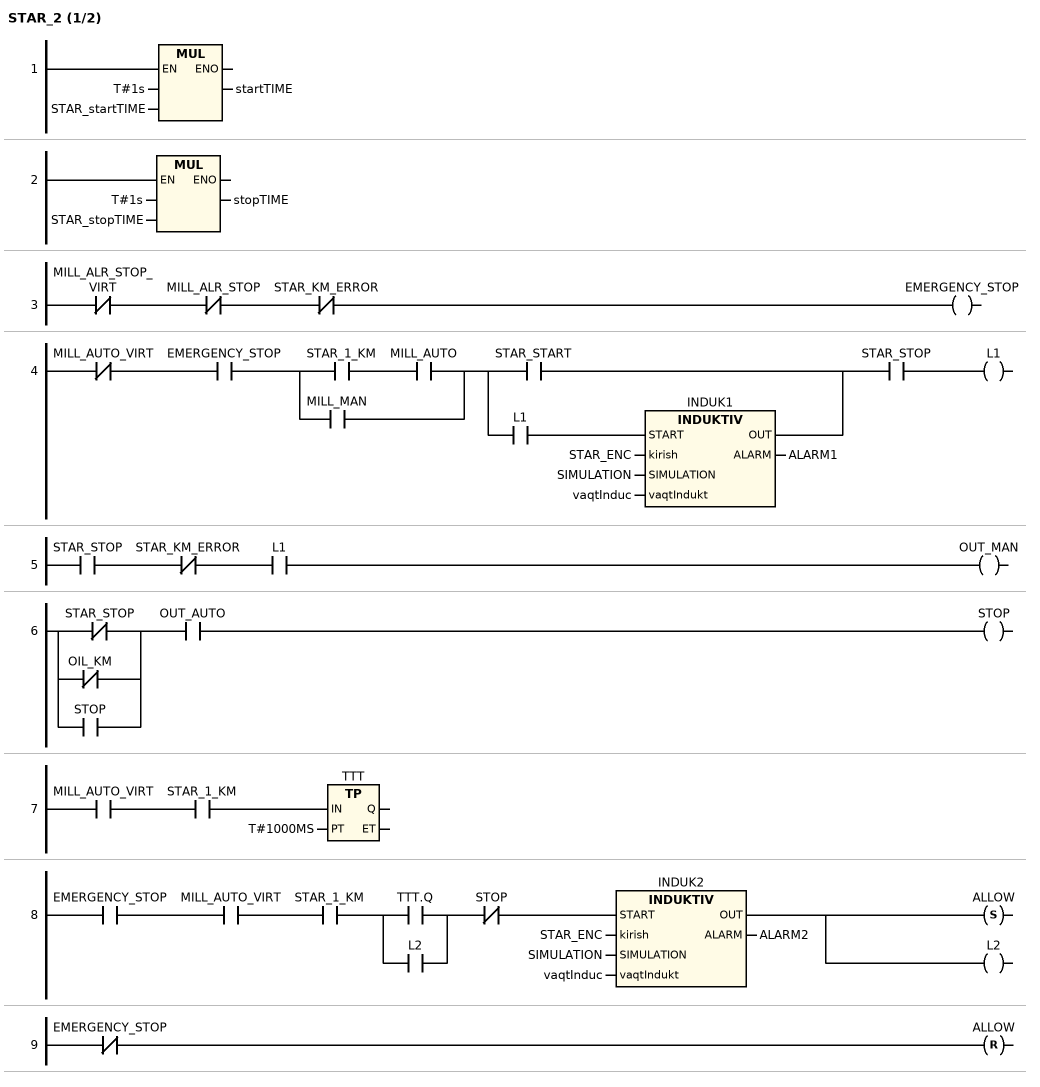
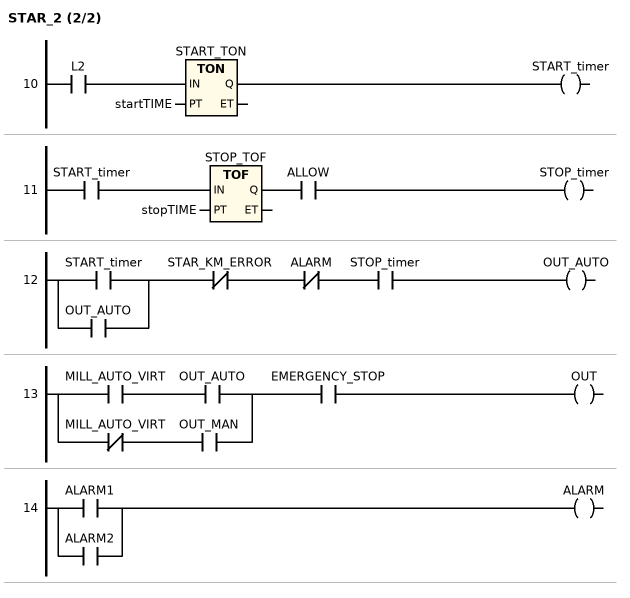
_LD_ (* Ladder Diagram *)
NETWORK 1
	*
		EN --- MUL(T#1s, STAR_startTIME) => startTIME
NETWORK 2
	*
		EN --- MUL(T#1s, STAR_stopTIME) => stopTIME
NETWORK 3
	[/MILL_ALR_STOP_VIRT] - [/MILL_ALR_STOP] - [/STAR_KM_ERROR] --- (EMERGENCY_STOP)
NETWORK 4
	[/MILL_AUTO_VIRT] - [EMERGENCY_STOP] - { [STAR_1_KM] - [MILL_AUTO] | [MILL_MAN] } - { [STAR_START] | [L1] - INDUK1:INDUKTIV(START: *, kirish: STAR_ENC, SIMULATION: SIMULATION, vaqtIndukt: vaqtInduc, ALARM => ALARM1) } - [STAR_STOP] --- (L1)
NETWORK 5
	[STAR_STOP] - [/STAR_KM_ERROR] - [L1] --- (OUT_MAN)
NETWORK 6
	{ [/STAR_STOP] | [/OIL_KM] | [STOP] } - [OUT_AUTO] --- (STOP)
NETWORK 7
	[MILL_AUTO_VIRT] - [STAR_1_KM] - TTT:TP(IN: *, PT: T#1000MS)
NETWORK 8
	[EMERGENCY_STOP] - [MILL_AUTO_VIRT] - [STAR_1_KM] - { [TTT.Q] | [L2] } - [/STOP] - INDUK2:INDUKTIV(START: *, kirish: STAR_ENC, SIMULATION: SIMULATION, vaqtIndukt: vaqtInduc, ALARM => ALARM2) --- (S ALLOW) (L2)
NETWORK 9
	[/EMERGENCY_STOP] --- (R ALLOW)
NETWORK 10
	[L2] - START_TON:TON(IN: *, PT: startTIME) --- (START_timer)
NETWORK 11
	[START_timer] - STOP_TOF:TOF(IN: *, PT: stopTIME) - [ALLOW] --- (STOP_timer)
NETWORK 12
	{ [START_timer] | [OUT_AUTO] } - [/STAR_KM_ERROR] - [/ALARM] - [STOP_timer] --- (OUT_AUTO)
NETWORK 13
	{ [MILL_AUTO_VIRT] - [OUT_AUTO] | [/MILL_AUTO_VIRT] - [OUT_MAN] } - [EMERGENCY_STOP] --- (OUT)
NETWORK 14
	{ [ALARM1] | [ALARM2] } --- (ALARM)
_END_LD_
(* the same logic as Structured Text *)
(* Network 1 *)
startTIME := T#1s * STAR_startTIME;
(* Network 2 *)
stopTIME := T#1s * STAR_stopTIME;
(* Network 3 *)
EMERGENCY_STOP := NOT MILL_ALR_STOP_VIRT AND NOT MILL_ALR_STOP AND NOT STAR_KM_ERROR;
(* Network 4 *)
_p1 := NOT MILL_AUTO_VIRT AND EMERGENCY_STOP AND (STAR_1_KM AND MILL_AUTO OR MILL_MAN);
INDUK1(START := _p1 AND L1, kirish := STAR_ENC, SIMULATION := SIMULATION, vaqtIndukt := vaqtInduc);
ALARM1 := INDUK1.ALARM;
L1 := (_p1 AND STAR_START OR INDUK1.OUT) AND STAR_STOP;
(* Network 5 *)
OUT_MAN := STAR_STOP AND NOT STAR_KM_ERROR AND L1;
(* Network 6 *)
STOP := (NOT STAR_STOP OR NOT OIL_KM OR STOP) AND OUT_AUTO;
(* Network 7 *)
TTT(IN := MILL_AUTO_VIRT AND STAR_1_KM, PT := T#1000MS);
(* Network 8 *)
INDUK2(START := EMERGENCY_STOP AND MILL_AUTO_VIRT AND STAR_1_KM AND (TTT.Q OR L2) AND NOT STOP, kirish := STAR_ENC, SIMULATION := SIMULATION, vaqtIndukt := vaqtInduc);
ALARM2 := INDUK2.ALARM;
IF INDUK2.OUT THEN ALLOW := TRUE; END_IF;
L2 := INDUK2.OUT;
(* Network 9 *)
IF NOT EMERGENCY_STOP THEN ALLOW := FALSE; END_IF;
(* Network 10 *)
START_TON(IN := L2, PT := startTIME);
START_timer := START_TON.Q;
(* Network 11 *)
STOP_TOF(IN := START_timer, PT := stopTIME);
STOP_timer := STOP_TOF.Q AND ALLOW;
(* Network 12 *)
OUT_AUTO := (START_timer OR OUT_AUTO) AND NOT STAR_KM_ERROR AND NOT ALARM AND STOP_timer;
(* Network 13 *)
OUT := (MILL_AUTO_VIRT AND OUT_AUTO OR NOT MILL_AUTO_VIRT AND OUT_MAN) AND EMERGENCY_STOP;
(* Network 14 *)
ALARM := ALARM1 OR ALARM2;
END_FUNCTION_BLOCK

(* POU SEP, LD *)
FUNCTION_BLOCK SEP
VAR_INPUT
	EN : BOOL;
	MILL_ALR_STOP: BOOL;
	MILL_ALR_STOP_VIRT : BOOL;
	MILL_AUTO : BOOL;
	MILL_AUTO_VIRT : BOOL;
	MILL_MAN : BOOL;
	SEPR_START : BOOL;
	SEPR_START_VIRT : BOOL;
	SEPR_ENC : BOOL;
	SEP_STOP : BOOL;


	SEP_KM_ERROR : BOOL;
	SIMULATION : BOOL := TRUE;
	vaqtInduc : WORD := 15;
	SEP_startTIME : WORD;
	SEP_stopTIME : WORD;
END_VAR

VAR_OUTPUT
	OUT : BOOL;
	ALARM : BOOL;
END_VAR
VAR
	INDUK1: INDUKTIV;
	INDUK2: INDUKTIV;
	OUT_MAN: BOOL;
	OUT_AUTO: BOOL;
	START_TON : TON;
	STOP_TOF : TOF;
	startTIME : TIME;
	stopTIME : TIME;
	L1: BOOL;
	L2: BOOL;
	ES: BOOL;
	EMERGENCY_STOP: BOOL;
	ALARM1 : BOOL;
	ALARM2 : BOOL;

	STOP: BOOL;
	ALLOW: BOOL;
	START_timer: BOOL;
	STOP_timer: BOOL;
END_VAR
VAR (* helpers for the ST form of the networks *)
	_p1 : BOOL;
END_VAR
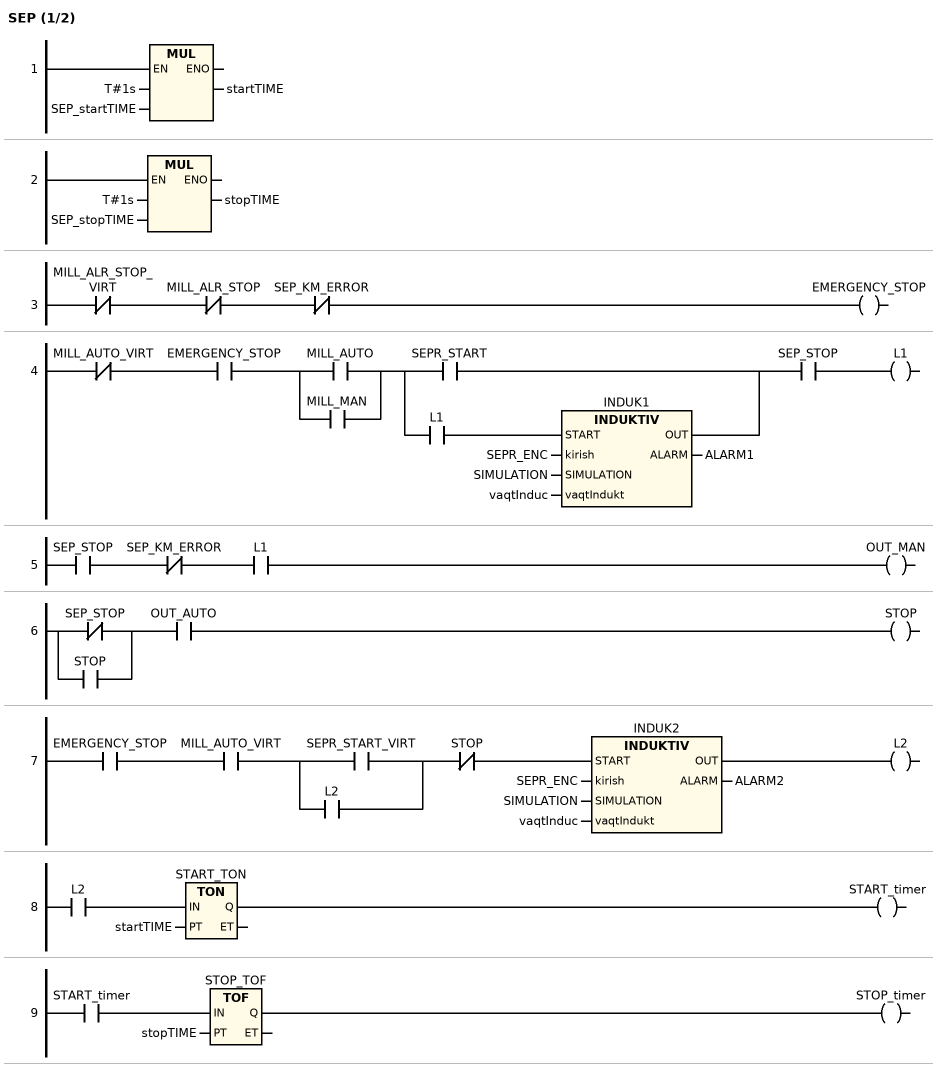
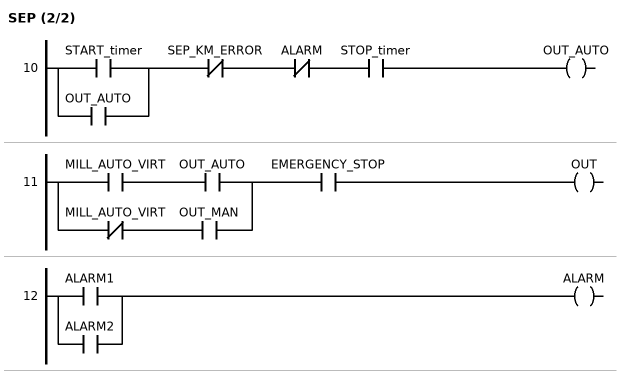
_LD_ (* Ladder Diagram *)
NETWORK 1
	*
		EN --- MUL(T#1s, SEP_startTIME) => startTIME
NETWORK 2
	*
		EN --- MUL(T#1s, SEP_stopTIME) => stopTIME
NETWORK 3
	[/MILL_ALR_STOP_VIRT] - [/MILL_ALR_STOP] - [/SEP_KM_ERROR] --- (EMERGENCY_STOP)
NETWORK 4
	[/MILL_AUTO_VIRT] - [EMERGENCY_STOP] - { [MILL_AUTO] | [MILL_MAN] } - { [SEPR_START] | [L1] - INDUK1:INDUKTIV(START: *, kirish: SEPR_ENC, SIMULATION: SIMULATION, vaqtIndukt: vaqtInduc, ALARM => ALARM1) } - [SEP_STOP] --- (L1)
NETWORK 5
	[SEP_STOP] - [/SEP_KM_ERROR] - [L1] --- (OUT_MAN)
NETWORK 6
	{ [/SEP_STOP] | [STOP] } - [OUT_AUTO] --- (STOP)
NETWORK 7
	[EMERGENCY_STOP] - [MILL_AUTO_VIRT] - { [SEPR_START_VIRT] | [L2] } - [/STOP] - INDUK2:INDUKTIV(START: *, kirish: SEPR_ENC, SIMULATION: SIMULATION, vaqtIndukt: vaqtInduc, ALARM => ALARM2) --- (L2)
NETWORK 8
	[L2] - START_TON:TON(IN: *, PT: startTIME) --- (START_timer)
NETWORK 9
	[START_timer] - STOP_TOF:TOF(IN: *, PT: stopTIME) --- (STOP_timer)
NETWORK 10
	{ [START_timer] | [OUT_AUTO] } - [/SEP_KM_ERROR] - [/ALARM] - [STOP_timer] --- (OUT_AUTO)
NETWORK 11
	{ [MILL_AUTO_VIRT] - [OUT_AUTO] | [/MILL_AUTO_VIRT] - [OUT_MAN] } - [EMERGENCY_STOP] --- (OUT)
NETWORK 12
	{ [ALARM1] | [ALARM2] } --- (ALARM)
_END_LD_
(* the same logic as Structured Text *)
(* Network 1 *)
startTIME := T#1s * SEP_startTIME;
(* Network 2 *)
stopTIME := T#1s * SEP_stopTIME;
(* Network 3 *)
EMERGENCY_STOP := NOT MILL_ALR_STOP_VIRT AND NOT MILL_ALR_STOP AND NOT SEP_KM_ERROR;
(* Network 4 *)
_p1 := NOT MILL_AUTO_VIRT AND EMERGENCY_STOP AND (MILL_AUTO OR MILL_MAN);
INDUK1(START := _p1 AND L1, kirish := SEPR_ENC, SIMULATION := SIMULATION, vaqtIndukt := vaqtInduc);
ALARM1 := INDUK1.ALARM;
L1 := (_p1 AND SEPR_START OR INDUK1.OUT) AND SEP_STOP;
(* Network 5 *)
OUT_MAN := SEP_STOP AND NOT SEP_KM_ERROR AND L1;
(* Network 6 *)
STOP := (NOT SEP_STOP OR STOP) AND OUT_AUTO;
(* Network 7 *)
INDUK2(START := EMERGENCY_STOP AND MILL_AUTO_VIRT AND (SEPR_START_VIRT OR L2) AND NOT STOP, kirish := SEPR_ENC, SIMULATION := SIMULATION, vaqtIndukt := vaqtInduc);
ALARM2 := INDUK2.ALARM;
L2 := INDUK2.OUT;
(* Network 8 *)
START_TON(IN := L2, PT := startTIME);
START_timer := START_TON.Q;
(* Network 9 *)
STOP_TOF(IN := START_timer, PT := stopTIME);
STOP_timer := STOP_TOF.Q;
(* Network 10 *)
OUT_AUTO := (START_timer OR OUT_AUTO) AND NOT SEP_KM_ERROR AND NOT ALARM AND STOP_timer;
(* Network 11 *)
OUT := (MILL_AUTO_VIRT AND OUT_AUTO OR NOT MILL_AUTO_VIRT AND OUT_MAN) AND EMERGENCY_STOP;
(* Network 12 *)
ALARM := ALARM1 OR ALARM2;
END_FUNCTION_BLOCK

(* POU OIL, LD *)
FUNCTION_BLOCK OIL
VAR_INPUT
	EN : BOOL;
	MILL_ALR_STOP: BOOL;
	MILL_ALR_STOP_VIRT : BOOL;
	MILL_AUTO : BOOL;
	MILL_AUTO_VIRT : BOOL;

	MILL_MAN : BOOL;
	OIL_START : BOOL;
	SEPR_RUN : BOOL;
	OIL_STOP : BOOL;
	MILL_KM : BOOL;
	OIL_KM_ERROR : BOOL;
	SEPR_START_VIRT : BOOL;

END_VAR

VAR_OUTPUT
	OUT : BOOL;
END_VAR
VAR
	INDUK1: INDUKTIV;
	INDUK2: INDUKTIV;
	OUT_MAN: BOOL;
	OUT_AUTO: BOOL;
	START_TON : TON;
	STOP_TOF : TOF;
	startTIME : TIME;
	stopTIME : TIME;
	L1: BOOL;
	L2: BOOL;
	ES: BOOL;
	EMERGENCY_STOP: BOOL;
	ALARM1 : BOOL;
	ALARM2 : BOOL;

	STOP: BOOL;
	ALLOW: BOOL;
	START_timer: BOOL;
	STOP_timer: BOOL;
	TTT : TP;
	L3: BOOL;
END_VAR
VAR (* helpers for the ST form of the networks *)
	_p1 : BOOL;
END_VAR
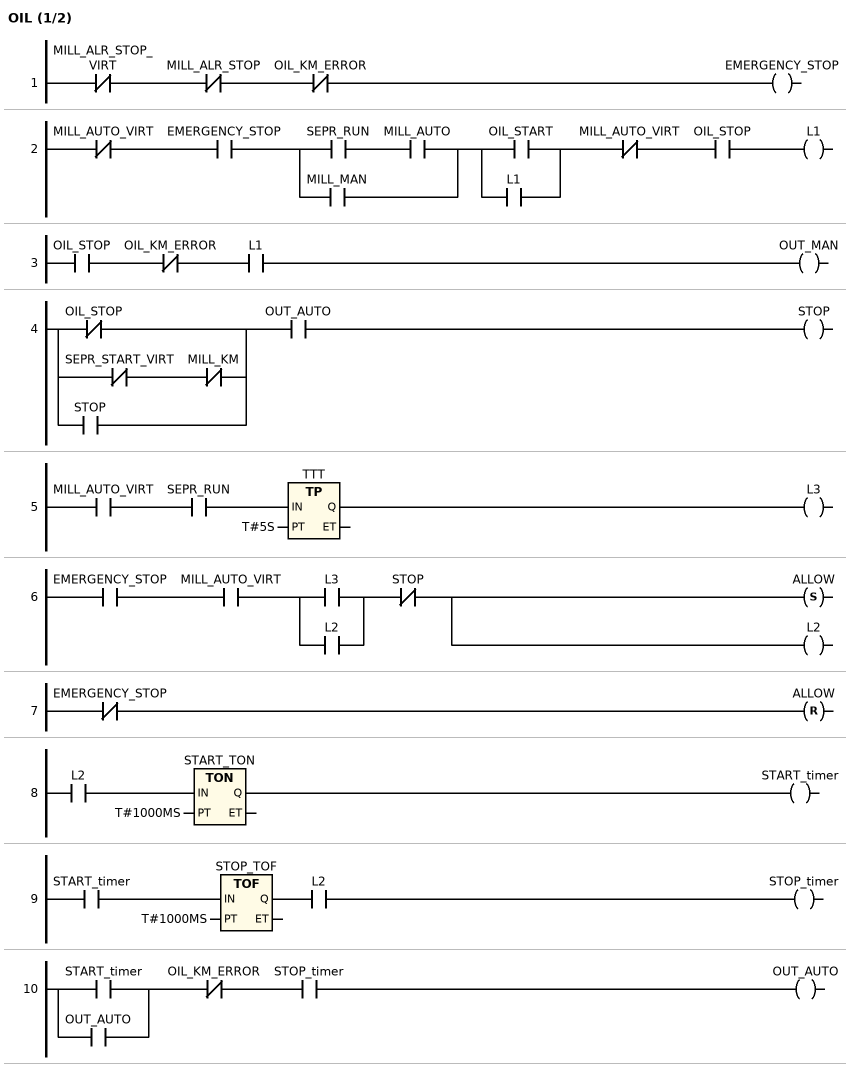
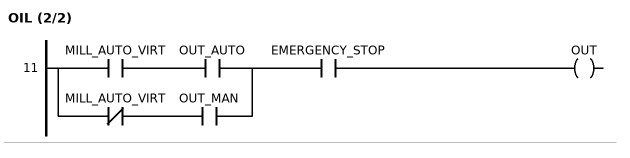
_LD_ (* Ladder Diagram *)
NETWORK 1
	[/MILL_ALR_STOP_VIRT] - [/MILL_ALR_STOP] - [/OIL_KM_ERROR] --- (EMERGENCY_STOP)
NETWORK 2
	[/MILL_AUTO_VIRT] - [EMERGENCY_STOP] - { [SEPR_RUN] - [MILL_AUTO] | [MILL_MAN] } - { [OIL_START] | [L1] } - [/MILL_AUTO_VIRT] - [OIL_STOP] --- (L1)
NETWORK 3
	[OIL_STOP] - [/OIL_KM_ERROR] - [L1] --- (OUT_MAN)
NETWORK 4
	{ [/OIL_STOP] | [/SEPR_START_VIRT] - [/MILL_KM] | [STOP] } - [OUT_AUTO] --- (STOP)
NETWORK 5
	[MILL_AUTO_VIRT] - [SEPR_RUN] - TTT:TP(IN: *, PT: T#5S) --- (L3)
NETWORK 6
	[EMERGENCY_STOP] - [MILL_AUTO_VIRT] - { [L3] | [L2] } - [/STOP] --- (S ALLOW) (L2)
NETWORK 7
	[/EMERGENCY_STOP] --- (R ALLOW)
NETWORK 8
	[L2] - START_TON:TON(IN: *, PT: T#1000MS) --- (START_timer)
NETWORK 9
	[START_timer] - STOP_TOF:TOF(IN: *, PT: T#1000MS) - [L2] --- (STOP_timer)
NETWORK 10
	{ [START_timer] | [OUT_AUTO] } - [/OIL_KM_ERROR] - [STOP_timer] --- (OUT_AUTO)
NETWORK 11
	{ [MILL_AUTO_VIRT] - [OUT_AUTO] | [/MILL_AUTO_VIRT] - [OUT_MAN] } - [EMERGENCY_STOP] --- (OUT)
_END_LD_
(* the same logic as Structured Text *)
(* Network 1 *)
EMERGENCY_STOP := NOT MILL_ALR_STOP_VIRT AND NOT MILL_ALR_STOP AND NOT OIL_KM_ERROR;
(* Network 2 *)
L1 := NOT MILL_AUTO_VIRT AND EMERGENCY_STOP AND (SEPR_RUN AND MILL_AUTO OR MILL_MAN) AND (OIL_START OR L1) AND NOT MILL_AUTO_VIRT AND OIL_STOP;
(* Network 3 *)
OUT_MAN := OIL_STOP AND NOT OIL_KM_ERROR AND L1;
(* Network 4 *)
STOP := (NOT OIL_STOP OR NOT SEPR_START_VIRT AND NOT MILL_KM OR STOP) AND OUT_AUTO;
(* Network 5 *)
TTT(IN := MILL_AUTO_VIRT AND SEPR_RUN, PT := T#5S);
L3 := TTT.Q;
(* Network 6 *)
_p1 := EMERGENCY_STOP AND MILL_AUTO_VIRT AND (L3 OR L2) AND NOT STOP;
IF _p1 THEN ALLOW := TRUE; END_IF;
L2 := _p1;
(* Network 7 *)
IF NOT EMERGENCY_STOP THEN ALLOW := FALSE; END_IF;
(* Network 8 *)
START_TON(IN := L2, PT := T#1000MS);
START_timer := START_TON.Q;
(* Network 9 *)
STOP_TOF(IN := START_timer, PT := T#1000MS);
STOP_timer := STOP_TOF.Q AND L2;
(* Network 10 *)
OUT_AUTO := (START_timer OR OUT_AUTO) AND NOT OIL_KM_ERROR AND STOP_timer;
(* Network 11 *)
OUT := (MILL_AUTO_VIRT AND OUT_AUTO OR NOT MILL_AUTO_VIRT AND OUT_MAN) AND EMERGENCY_STOP;
END_FUNCTION_BLOCK

(* POU MILL, LD *)
FUNCTION_BLOCK MILL
VAR_INPUT
	EN : BOOL;
	MILL_ALR_STOP: BOOL;
	MILL_ALR_STOP_VIRT : BOOL;
	MILL_AUTO : BOOL;
	MILL_AUTO_VIRT : BOOL;
	MILL_MAN : BOOL;
	MILL_START : BOOL;
	OIL_KM : BOOL;
	MILL_ENC : BOOL;
	MILL_STOP : BOOL;
	FAN_KM : BOOL;
	MILL_KM_ERROR : BOOL;
	SIMULATION : BOOL := TRUE;
	SEPR_START_VIRT : BOOL;
	vaqtInduc : WORD := 15;
	MILL_startTIME : WORD;
	MILL_stopTIME : WORD;
	SEP_KM : BOOL;
END_VAR

VAR_OUTPUT
	OUT : BOOL;
	ALARM : BOOL;
END_VAR
VAR
	INDUK1: INDUKTIV;
	INDUK2: INDUKTIV;
	OUT_MAN: BOOL;
	OUT_AUTO: BOOL;
	START_TON : TON;
	STOP_TOF : TOF;
	startTIME : TIME;
	stopTIME : TIME;
	L1: BOOL;
	L2: BOOL;
	ES: BOOL;
	EMERGENCY_STOP: BOOL;
	ALARM1 : BOOL;
	ALARM2 : BOOL;

	STOP: BOOL;
	ALLOW: BOOL;
	START_timer: BOOL;
	STOP_timer: BOOL;
	TTT : TP;
	STOP_I: BOOL;
END_VAR
VAR (* helpers for the ST form of the networks *)
	_p1 : BOOL;
	_p2 : BOOL;
END_VAR
